LIN {X 0,Y 305.488,Z 300.056,A -85,B 0,C 180,E1 -15819.813,E2 -15819.813} C_VEL
LIN {X 0,Y 305.533,Z 300.043,A -85,B 0,C 180,E1 -15822.6,E2 -15822.6} C_VEL
LIN {X 0,Y 305.618,Z 300.037,A -85,B 0,C 180,E1 -15825.347,E2 -15825.347} C_VEL
LIN {X 0,Y 305.615,Z 300.039,A -85,B 0,C 180,E1 -15829.399,E2 -15829.399} C_VEL
LIN {X 0,Y 305.761,Z 300.017,A -85,B 0,C 180,E1 -15832.073,E2 -15832.073} C_VEL
LIN {X 0,Y 305.66,Z 300.028,A -85,B 0,C 180,E1 -15834.723,E2 -15834.723} C_VEL
LIN {X 0,Y 305.94,Z 299.998,A -85,B 0,C 180,E1 -15838.684,E2 -15838.684} C_VEL
LIN {X 0,Y 305.938,Z 299.999,A -85,B 0,C 180,E1 -15841.316,E2 -15841.316} C_VEL
LIN {X 0,Y 305.788,Z 300.021,A -85,B 0,C 180,E1 -15846.599,E2 -15846.599} C_VEL
LIN {X 0,Y 305.685,Z 300.023,A -85,B 0,C 180,E1 -15849.261,E2 -15849.261} C_VEL
LIN {X 0,Y 305.575,Z 300.037,A -85,B 0,C 180,E1 -15853.296,E2 -15853.296} C_VEL
LIN {X 0,Y 305.542,Z 300.054,A -85,B 0,C 180,E1 -15856.023,E2 -15856.023} C_VEL
LIN {X 0,Y 305.475,Z 300.064,A -85,B 0,C 180,E1 -15860.188,E2 -15860.188} C_VEL
LIN {X 0,Y 305.447,Z 300.063,A -85,B 0,C 180,E1 -15864.466,E2 -15864.466} C_VEL
LIN {X 0,Y 305.444,Z 300.063,A -85,B 0,C 180,E1 -15867.399,E2 -15867.399} C_VEL
LIN {X 0,Y 305.423,Z 300.065,A -85,B 0,C 180,E1 -15870.413,E2 -15870.413} C_VEL
LIN {X 0,Y 305.457,Z 300.057,A -85,B 0,C 180,E1 -15874.079,E2 -15874.079} C_VEL
LIN {X 0,Y 305.446,Z 300.057,A -85,B 0,C 180,E1 -15876.743,E2 -15876.743} C_VEL
LIN {X 0,Y 305.403,Z 300.042,A -85,B 0,C 180,E1 -15880.59,E2 -15880.59} C_VEL
LIN {X 0,Y 305.415,Z 300.065,A -85,B 0,C 180,E1 -15883.657,E2 -15883.657} C_VEL
LIN {X 0,Y 305.407,Z 300.074,A -85,B 0,C 180,E1 -15886.973,E2 -15886.973} C_VEL
LIN {X 0,Y 308.846,Z 311.457,A -85,B 0,C 180,E1 -15890.686,E2 -15890.686} C_VEL
LIN {X 0,Y 309.648,Z 314.272,A -85,B 0,C 180,E1 -15891.522,E2 -15891.522} C_VEL
LIN {X 0,Y 318.82,Z 331.707,A -85,B 0,C 180,E1 -15893.292,E2 -15893.292} C_VEL
LIN {X 0,Y 326.748,Z 348.767,A -85,B 0,C 180,E1 -15894.765,E2 -15894.765} C_VEL
LIN {X 0,Y 329.337,Z 355.038,A -85,B 0,C 180,E1 -15895.243,E2 -15895.243} C_VEL
LIN {X 0,Y 331.45,Z 367.704,A -85,B 0,C 180,E1 -15895.82,E2 -15895.82} C_VEL
LIN {X 0,Y 328.353,Z 458.786,A -85,B 0,C 180,E1 -15897.787,E2 -15897.787} C_VEL
LIN {X 0,Y 327.344,Z 483.079,A -85,B 0,C 180,E1 -15898.355,E2 -15898.355} C_VEL
LIN {X 0,Y 326.05,Z 498.482,A -85,B 0,C 180,E1 -15898.939,E2 -15898.939} C_VEL
LIN {X 0,Y 324.286,Z 513.373,A -85,B 0,C 180,E1 -15899.744,E2 -15899.744} C_VEL
LIN {X 0,Y 322.3,Z 527.368,A -85,B 0,C 180,E1 -15900.754,E2 -15900.754} C_VEL
LIN {X 0,Y 320.028,Z 540.986,A -85,B 0,C 180,E1 -15902.005,E2 -15902.005} C_VEL
LIN {X 0,Y 317.409,Z 554.417,A -85,B 0,C 180,E1 -15903.539,E2 -15903.539} C_VEL
LIN {X 0,Y 314.806,Z 566.654,A -85,B 0,C 180,E1 -15905.255,E2 -15905.255} C_VEL
LIN {X 0,Y 312.33,Z 578.002,A -85,B 0,C 180,E1 -15907.196,E2 -15907.196} C_VEL
LIN {X 0,Y 310.016,Z 588.691,A -85,B 0,C 180,E1 -15909.429,E2 -15909.429} C_VEL
LIN {X 0,Y 307.942,Z 597.734,A -85,B 0,C 180,E1 -15911.712,E2 -15911.712} C_VEL
LIN {X 0,Y 306.367,Z 605.243,A -85,B 0,C 180,E1 -15914.022,E2 -15914.022} C_VEL
LIN {X 0,Y 305.088,Z 612.254,A -85,B 0,C 180,E1 -15916.682,E2 -15916.682} C_VEL
LIN {X 0,Y 304.181,Z 617.769,A -85,B 0,C 180,E1 -15919.349,E2 -15919.349} C_VEL
LIN {X 0,Y 303.767,Z 621.945,A -85,B 0,C 180,E1 -15922.021,E2 -15922.021} C_VEL
LIN {X 0,Y 303.596,Z 624.875,A -85,B 0,C 180,E1 -15924.687,E2 -15924.687} C_VEL
LIN {X 0,Y 303.592,Z 626.624,A -85,B 0,C 180,E1 -15927.346,E2 -15927.346} C_VEL
LIN {X 0,Y 303.602,Z 627.222,A -85,B 0,C 180,E1 -15930,E2 -15930} C_VEL
LIN {X 0,Y 303.591,Z 626.615,A -85,B 0,C 180,E1 -15932.654,E2 -15932.654} C_VEL
LIN {X 0,Y 303.624,Z 624.655,A -85,B 0,C 180,E1 -15935.544,E2 -15935.544} C_VEL
LIN {X 0,Y 303.765,Z 621.916,A -85,B 0,C 180,E1 -15937.979,E2 -15937.979} C_VEL
LIN {X 0,Y 304.18,Z 617.735,A -85,B 0,C 180,E1 -15940.651,E2 -15940.651} C_VEL
LIN {X 0,Y 305.08,Z 612.205,A -85,B 0,C 180,E1 -15943.318,E2 -15943.318} C_VEL
LIN {X 0,Y 306.362,Z 605.173,A -85,B 0,C 180,E1 -15945.978,E2 -15945.978} C_VEL
LIN {X 0,Y 308.205,Z 596.433,A -85,B 0,C 180,E1 -15948.617,E2 -15948.617} C_VEL
LIN {X 0,Y 310.357,Z 587.156,A -85,B 0,C 180,E1 -15950.894,E2 -15950.894} C_VEL
LIN {X 0,Y 312.379,Z 577.896,A -85,B 0,C 180,E1 -15952.8,E2 -15952.8} C_VEL
LIN {X 0,Y 314.82,Z 566.53,A -85,B 0,C 180,E1 -15954.744,E2 -15954.744} C_VEL
LIN {X 0,Y 317.413,Z 554.269,A -85,B 0,C 180,E1 -15956.461,E2 -15956.461} C_VEL
LIN {X 0,Y 320.015,Z 540.79,A -85,B 0,C 180,E1 -15957.996,E2 -15957.996} C_VEL
LIN {X 0,Y 322.452,Z 526.115,A -85,B 0,C 180,E1 -15959.33,E2 -15959.33} C_VEL
LIN {X 0,Y 324.573,Z 510.682,A -85,B 0,C 180,E1 -15960.406,E2 -15960.406} C_VEL
LIN {X 0,Y 326.261,Z 495.632,A -85,B 0,C 180,E1 -15961.174,E2 -15961.174} C_VEL
LIN {X 0,Y 327.451,Z 479.865,A -85,B 0,C 180,E1 -15961.724,E2 -15961.724} C_VEL
LIN {X 0,Y 330.751,Z 387.93,A -85,B 0,C 180,E1 -15963.718,E2 -15963.718} C_VEL
LIN {X 0,Y 331.325,Z 367.172,A -85,B 0,C 180,E1 -15964.182,E2 -15964.182} C_VEL
LIN {X 0,Y 328.976,Z 353.98,A -85,B 0,C 180,E1 -15964.8,E2 -15964.8} C_VEL
LIN {X 0,Y 320.543,Z 335.198,A -85,B 0,C 180,E1 -15966.354,E2 -15966.354} C_VEL
LIN {X 0,Y 311.857,Z 318.359,A -85,B 0,C 180,E1 -15968.007,E2 -15968.007} C_VEL
LIN {X 0,Y 309.559,Z 314.082,A -85,B 0,C 180,E1 -15968.469,E2 -15968.469} C_VEL
LIN {X 0,Y 306.242,Z 302.692,A -85,B 0,C 180,E1 -15972.101,E2 -15972.101} C_VEL
LIN {X 0,Y 305.408,Z 300.068,A -85,B 0,C 180,E1 -15973.027,E2 -15973.027} C_VEL
LIN {X 0,Y 305.429,Z 300.063,A -85,B 0,C 180,E1 -15977.418,E2 -15977.418} C_VEL
LIN {X 0,Y 305.439,Z 300.06,A -85,B 0,C 180,E1 -15981.592,E2 -15981.592} C_VEL
LIN {X 0,Y 305.453,Z 300.057,A -85,B 0,C 180,E1 -15984.886,E2 -15984.886} C_VEL
LIN {X 0,Y 305.434,Z 300.063,A -85,B 0,C 180,E1 -15988.358,E2 -15988.358} C_VEL
LIN {X 0,Y 305.467,Z 300.058,A -85,B 0,C 180,E1 -15991.108,E2 -15991.108} C_VEL
LIN {X 0,Y 305.472,Z 300.06,A -85,B 0,C 180,E1 -15994.079,E2 -15994.079} C_VEL
LIN {X 0,Y 305.455,Z 300.059,A -85,B 0,C 180,E1 -15998.4,E2 -15998.4} C_VEL
LIN {X 0,Y 305.529,Z 300.035,A -85,B 0,C 180,E1 -16002.6,E2 -16002.6} C_VEL
LIN {X 0,Y 305.618,Z 300.04,A -85,B 0,C 180,E1 -16005.348,E2 -16005.348} C_VEL
LIN {X 0,Y 305.612,Z 300.009,A -85,B 0,C 180,E1 -16009.399,E2 -16009.399} C_VEL
LIN {X 0,Y 305.732,Z 300.027,A -85,B 0,C 180,E1 -16012.072,E2 -16012.072} C_VEL
LIN {X 0,Y 305.651,Z 300.027,A -85,B 0,C 180,E1 -16014.723,E2 -16014.723} C_VEL
LIN {X 0,Y 305.938,Z 299.991,A -85,B 0,C 180,E1 -16018.684,E2 -16018.684} C_VEL
LIN {X 0,Y 305.926,Z 300.001,A -85,B 0,C 180,E1 -16021.317,E2 -16021.317} C_VEL
LIN {X 0,Y 305.658,Z 300.036,A -85,B 0,C 180,E1 -16025.277,E2 -16025.277} C_VEL
LIN {X 0,Y 305.753,Z 300.023,A -85,B 0,C 180,E1 -16027.927,E2 -16027.927} C_VEL
LIN {X 0,Y 305.588,Z 300.043,A -85,B 0,C 180,E1 -16031.946,E2 -16031.946} C_VEL
LIN {X 0,Y 305.6,Z 300.036,A -85,B 0,C 180,E1 -16035.014,E2 -16035.014} C_VEL
LIN {X 0,Y 305.509,Z 300.039,A -85,B 0,C 180,E1 -16038.788,E2 -16038.788} C_VEL
LIN {X 0,Y 305.479,Z 300.052,A -85,B 0,C 180,E1 -16043.04,E2 -16043.04} C_VEL
LIN {X 0,Y 305.497,Z 300.038,A -85,B 0,C 180,E1 -16046.211,E2 -16046.211} C_VEL
LIN {X 0,Y 305.478,Z 300.046,A -85,B 0,C 180,E1 -16049.047,E2 -16049.047} C_VEL
LIN {X 0,Y 305.436,Z 300.057,A -85,B 0,C 180,E1 -16051.953,E2 -16051.953} C_VEL
LIN {X 0,Y 305.455,Z 300.057,A -85,B 0,C 180,E1 -16055.114,E2 -16055.114} C_VEL
LIN {X 0,Y 305.434,Z 300.061,A -85,B 0,C 180,E1 -16058.527,E2 -16058.527} C_VEL
LIN {X 0,Y 305.45,Z 300.058,A -85,B 0,C 180,E1 -16062.587,E2 -16062.587} C_VEL
LIN {X 0,Y 305.421,Z 300.065,A -85,B 0,C 180,E1 -16066.346,E2 -16066.346} C_VEL
LIN {X 0,Y 305.455,Z 300.061,A -85,B 0,C 180,E1 -16069.893,E2 -16069.893} C_VEL
LIN {X 0,Y 305.446,Z 300.076,A -85,B 0,C 180,E1 -16070.761,E2 -16070.761} C_VEL
LIN {X 0,Y 305.611,Z 300.81,A -85,B 0,C 180,E1 -16071.007,E2 -16071.007} C_VEL
LIN {X 0,Y 306.858,Z 303.478,A -85,B 0,C 180,E1 -16071.275,E2 -16071.275} C_VEL
LIN {X 0,Y 308.864,Z 306.49,A -85,B 0,C 180,E1 -16071.663,E2 -16071.663} C_VEL
LIN {X 0,Y 314.538,Z 316.113,A -85,B 0,C 180,E1 -16072.754,E2 -16072.754} C_VEL
LIN {X 0,Y 323.344,Z 332.892,A -85,B 0,C 180,E1 -16074.393,E2 -16074.393} C_VEL
LIN {X 0,Y 331.832,Z 351.222,A -85,B 0,C 180,E1 -16075.916,E2 -16075.916} C_VEL
LIN {X 0,Y 329.184,Z 429.846,A -85,B 0,C 180,E1 -16077.619,E2 -16077.619} C_VEL
LIN {X 0,Y 327.853,Z 465.342,A -85,B 0,C 180,E1 -16078.41,E2 -16078.41} C_VEL
LIN {X 0,Y 326.688,Z 481.055,A -85,B 0,C 180,E1 -16078.99,E2 -16078.99} C_VEL
LIN {X 0,Y 325.166,Z 496.001,A -85,B 0,C 180,E1 -16079.798,E2 -16079.798} C_VEL
LIN {X 0,Y 323.552,Z 509.183,A -85,B 0,C 180,E1 -16080.75,E2 -16080.75} C_VEL
LIN {X 0,Y 321.363,Z 522.677,A -85,B 0,C 180,E1 -16081.954,E2 -16081.954} C_VEL
LIN {X 0,Y 319.149,Z 535.149,A -85,B 0,C 180,E1 -16083.342,E2 -16083.342} C_VEL
LIN {X 0,Y 316.521,Z 547.786,A -85,B 0,C 180,E1 -16085.048,E2 -16085.048} C_VEL
LIN {X 0,Y 314.516,Z 557.561,A -85,B 0,C 180,E1 -16086.652,E2 -16086.652} C_VEL
LIN {X 0,Y 312.254,Z 567.396,A -85,B 0,C 180,E1 -16088.547,E2 -16088.547} C_VEL
LIN {X 0,Y 310.023,Z 577.09,A -85,B 0,C 180,E1 -16090.81,E2 -16090.81} C_VEL
LIN {X 0,Y 308.026,Z 585.389,A -85,B 0,C 180,E1 -16093.163,E2 -16093.163} C_VEL
LIN {X 0,Y 306.706,Z 591.827,A -85,B 0,C 180,E1 -16095.401,E2 -16095.401} C_VEL
LIN {X 0,Y 305.372,Z 597.993,A -85,B 0,C 180,E1 -16098.046,E2 -16098.046} C_VEL
LIN {X 0,Y 304.57,Z 602.747,A -85,B 0,C 180,E1 -16100.705,E2 -16100.705} C_VEL
LIN {X 0,Y 304.046,Z 606.228,A -85,B 0,C 180,E1 -16103.363,E2 -16103.363} C_VEL
LIN {X 0,Y 303.789,Z 608.528,A -85,B 0,C 180,E1 -16106.02,E2 -16106.02} C_VEL
LIN {X 0,Y 303.608,Z 609.703,A -85,B 0,C 180,E1 -16108.674,E2 -16108.674} C_VEL
LIN {X 0,Y 303.608,Z 609.717,A -85,B 0,C 180,E1 -16111.326,E2 -16111.326} C_VEL
LIN {X 0,Y 303.781,Z 608.598,A -85,B 0,C 180,E1 -16113.98,E2 -16113.98} C_VEL
LIN {X 0,Y 304.041,Z 606.352,A -85,B 0,C 180,E1 -16116.637,E2 -16116.637} C_VEL
LIN {X 0,Y 304.55,Z 602.921,A -85,B 0,C 180,E1 -16119.296,E2 -16119.296} C_VEL
LIN {X 0,Y 305.337,Z 598.223,A -85,B 0,C 180,E1 -16121.955,E2 -16121.955} C_VEL
LIN {X 0,Y 306.679,Z 592.126,A -85,B 0,C 180,E1 -16124.6,E2 -16124.6} C_VEL
LIN {X 0,Y 308.302,Z 584.452,A -85,B 0,C 180,E1 -16127.238,E2 -16127.238} C_VEL
LIN {X 0,Y 310.219,Z 576.262,A -85,B 0,C 180,E1 -16129.521,E2 -16129.521} C_VEL
LIN {X 0,Y 312.519,Z 566.392,A -85,B 0,C 180,E1 -16131.78,E2 -16131.78} C_VEL
LIN {X 0,Y 314.726,Z 556.192,A -85,B 0,C 180,E1 -16133.715,E2 -16133.715} C_VEL
LIN {X 0,Y 317.365,Z 544.212,A -85,B 0,C 180,E1 -16135.583,E2 -16135.583} C_VEL
LIN {X 0,Y 319.716,Z 532.118,A -85,B 0,C 180,E1 -16137.137,E2 -16137.137} C_VEL
LIN {X 0,Y 322.078,Z 518.969,A -85,B 0,C 180,E1 -16138.51,E2 -16138.51} C_VEL
LIN {X 0,Y 324.033,Z 505.698,A -85,B 0,C 180,E1 -16139.632,E2 -16139.632} C_VEL
LIN {X 0,Y 325.667,Z 491.769,A -85,B 0,C 180,E1 -16140.561,E2 -16140.561} C_VEL
LIN {X 0,Y 327.101,Z 476.492,A -85,B 0,C 180,E1 -16141.31,E2 -16141.31} C_VEL
LIN {X 0,Y 328.115,Z 461.755,A -85,B 0,C 180,E1 -16141.787,E2 -16141.787} C_VEL
LIN {X 0,Y 331.406,Z 368.205,A -85,B 0,C 180,E1 -16143.815,E2 -16143.815} C_VEL
LIN {X 0,Y 331.011,Z 364.38,A -85,B 0,C 180,E1 -16143.96,E2 -16143.96} C_VEL
LIN {X 0,Y 329.874,Z 360.802,A -85,B 0,C 180,E1 -16144.186,E2 -16144.186} C_VEL
LIN {X 0,Y 324.321,Z 349.64,A -85,B 0,C 180,E1 -16145.156,E2 -16145.156} C_VEL
LIN {X 0,Y 316.974,Z 334.175,A -85,B 0,C 180,E1 -16146.53,E2 -16146.53} C_VEL
LIN {X 0,Y 309.997,Z 320.812,A -85,B 0,C 180,E1 -16147.881,E2 -16147.881} C_VEL
LIN {X 0,Y 303.322,Z 309.395,A -85,B 0,C 180,E1 -16149.217,E2 -16149.217} C_VEL
LIN {X 0,Y 301.13,Z 305.909,A -85,B 0,C 180,E1 -16149.667,E2 -16149.667} C_VEL
LIN {X 0,Y 298.982,Z 302.953,A -85,B 0,C 180,E1 -16150.102,E2 -16150.102} C_VEL
LIN {X 0,Y 298.409,Z 300.93,A -85,B 0,C 180,E1 -16150.301,E2 -16150.301} C_VEL
LIN {X 0,Y 298.396,Z 300.94,A -85,B 0,C 180,E1 -16153.102,E2 -16153.102} C_VEL
LIN {X 0,Y 298.399,Z 300.931,A -85,B 0,C 180,E1 -16156.92,E2 -16156.92} C_VEL
LIN {X 0,Y 298.393,Z 300.941,A -85,B 0,C 180,E1 -16161.007,E2 -16161.007} C_VEL
LIN {X 0,Y 298.399,Z 300.919,A -85,B 0,C 180,E1 -16163.927,E2 -16163.927} C_VEL
LIN {X 0,Y 298.387,Z 300.935,A -85,B 0,C 180,E1 -16167.199,E2 -16167.199} C_VEL
LIN {X 0,Y 298.408,Z 300.919,A -85,B 0,C 180,E1 -16170.62,E2 -16170.62} C_VEL
LIN {X 0,Y 298.438,Z 300.932,A -85,B 0,C 180,E1 -16173.489,E2 -16173.489} C_VEL
LIN {X 0,Y 298.422,Z 300.939,A -85,B 0,C 180,E1 -16176.7,E2 -16176.7} C_VEL
LIN {X 0,Y 298.496,Z 300.929,A -85,B 0,C 180,E1 -16180.754,E2 -16180.754} C_VEL
LIN {X 0,Y 298.579,Z 300.917,A -85,B 0,C 180,E1 -16184.994,E2 -16184.994} C_VEL
LIN {X 0,Y 298.574,Z 300.918,A -85,B 0,C 180,E1 -16189.146,E2 -16189.146} C_VEL
LIN {X 0,Y 298.708,Z 300.896,A -85,B 0,C 180,E1 -16191.884,E2 -16191.884} C_VEL
LIN {X 0,Y 298.63,Z 300.905,A -85,B 0,C 180,E1 -16194.598,E2 -16194.598} C_VEL
LIN {X 0,Y 298.907,Z 300.874,A -85,B 0,C 180,E1 -16198.653,E2 -16198.653} C_VEL
LIN {X 0,Y 298.905,Z 300.875,A -85,B 0,C 180,E1 -16201.347,E2 -16201.347} C_VEL
LIN {X 0,Y 298.737,Z 300.901,A -85,B 0,C 180,E1 -16206.755,E2 -16206.755} C_VEL
LIN {X 0,Y 298.616,Z 300.904,A -85,B 0,C 180,E1 -16209.482,E2 -16209.482} C_VEL
LIN {X 0,Y 298.534,Z 300.914,A -85,B 0,C 180,E1 -16213.616,E2 -16213.616} C_VEL
LIN {X 0,Y 298.475,Z 300.931,A -85,B 0,C 180,E1 -16216.413,E2 -16216.413} C_VEL
LIN {X 0,Y 298.433,Z 300.938,A -85,B 0,C 180,E1 -16219.617,E2 -16219.617} C_VEL
LIN {X 0,Y 298.38,Z 300.944,A -85,B 0,C 180,E1 -16223.604,E2 -16223.604} C_VEL
LIN {X 0,Y 298.395,Z 300.936,A -85,B 0,C 180,E1 -16226.583,E2 -16226.583} C_VEL
LIN {X 0,Y 298.386,Z 300.943,A -85,B 0,C 180,E1 -16229.645,E2 -16229.645} C_VEL
LIN {X 0,Y 298.385,Z 300.933,A -85,B 0,C 180,E1 -16232.801,E2 -16232.801} C_VEL
LIN {X 0,Y 298.42,Z 300.932,A -85,B 0,C 180,E1 -16236.803,E2 -16236.803} C_VEL
LIN {X 0,Y 298.341,Z 300.923,A -85,B 0,C 180,E1 -16241.269,E2 -16241.269} C_VEL
LIN {X 0,Y 298.35,Z 300.947,A -85,B 0,C 180,E1 -16245.036,E2 -16245.036} C_VEL
LIN {X 0,Y 298.373,Z 300.96,A -85,B 0,C 180,E1 -16246.044,E2 -16246.044} C_VEL
LIN {X 0,Y 301.739,Z 312.035,A -85,B 0,C 180,E1 -16249.807,E2 -16249.807} C_VEL
LIN {X 0,Y 302.287,Z 313.971,A -85,B 0,C 180,E1 -16250.402,E2 -16250.402} C_VEL
LIN {X 0,Y 310.364,Z 328.922,A -85,B 0,C 180,E1 -16252.047,E2 -16252.047} C_VEL
LIN {X 0,Y 318.508,Z 345.475,A -85,B 0,C 180,E1 -16253.628,E2 -16253.628} C_VEL
LIN {X 0,Y 323.829,Z 358.27,A -85,B 0,C 180,E1 -16254.655,E2 -16254.655} C_VEL
LIN {X 0,Y 325.57,Z 369.904,A -85,B 0,C 180,E1 -16255.177,E2 -16255.177} C_VEL
LIN {X 0,Y 321.691,Z 476.003,A -85,B 0,C 180,E1 -16257.501,E2 -16257.501} C_VEL
LIN {X 0,Y 320.646,Z 491.352,A -85,B 0,C 180,E1 -16257.986,E2 -16257.986} C_VEL
LIN {X 0,Y 319.142,Z 505.626,A -85,B 0,C 180,E1 -16258.651,E2 -16258.651} C_VEL
LIN {X 0,Y 317.264,Z 519.739,A -85,B 0,C 180,E1 -16259.547,E2 -16259.547} C_VEL
LIN {X 0,Y 315.181,Z 532.909,A -85,B 0,C 180,E1 -16260.623,E2 -16260.623} C_VEL
LIN {X 0,Y 312.612,Z 546.5,A -85,B 0,C 180,E1 -16262.012,E2 -16262.012} C_VEL
LIN {X 0,Y 310.005,Z 558.926,A -85,B 0,C 180,E1 -16263.583,E2 -16263.583} C_VEL
LIN {X 0,Y 307.417,Z 570.373,A -85,B 0,C 180,E1 -16265.341,E2 -16265.341} C_VEL
LIN {X 0,Y 304.917,Z 581.187,A -85,B 0,C 180,E1 -16267.352,E2 -16267.352} C_VEL
LIN {X 0,Y 302.975,Z 589.85,A -85,B 0,C 180,E1 -16269.284,E2 -16269.284} C_VEL
LIN {X 0,Y 300.864,Z 598.656,A -85,B 0,C 180,E1 -16271.619,E2 -16271.619} C_VEL
LIN {X 0,Y 299.142,Z 606.68,A -85,B 0,C 180,E1 -16274.234,E2 -16274.234} C_VEL
LIN {X 0,Y 297.858,Z 613.546,A -85,B 0,C 180,E1 -16277.047,E2 -16277.047} C_VEL
LIN {X 0,Y 297.019,Z 618.735,A -85,B 0,C 180,E1 -16279.778,E2 -16279.778} C_VEL
LIN {X 0,Y 296.694,Z 621.742,A -85,B 0,C 180,E1 -16281.829,E2 -16281.829} C_VEL
LIN {X 0,Y 296.511,Z 624.672,A -85,B 0,C 180,E1 -16284.56,E2 -16284.56} C_VEL
LIN {X 0,Y 296.516,Z 626.422,A -85,B 0,C 180,E1 -16287.283,E2 -16287.283} C_VEL
LIN {X 0,Y 296.517,Z 627.019,A -85,B 0,C 180,E1 -16290,E2 -16290} C_VEL
LIN {X 0,Y 296.515,Z 626.412,A -85,B 0,C 180,E1 -16292.717,E2 -16292.717} C_VEL
LIN {X 0,Y 296.511,Z 624.65,A -85,B 0,C 180,E1 -16295.44,E2 -16295.44} C_VEL
LIN {X 0,Y 296.691,Z 621.711,A -85,B 0,C 180,E1 -16298.171,E2 -16298.171} C_VEL
LIN {X 0,Y 297.142,Z 617.529,A -85,B 0,C 180,E1 -16300.907,E2 -16300.907} C_VEL
LIN {X 0,Y 298.089,Z 611.998,A -85,B 0,C 180,E1 -16303.637,E2 -16303.637} C_VEL
LIN {X 0,Y 299.481,Z 604.967,A -85,B 0,C 180,E1 -16306.356,E2 -16306.356} C_VEL
LIN {X 0,Y 301.407,Z 596.226,A -85,B 0,C 180,E1 -16309.052,E2 -16309.052} C_VEL
LIN {X 0,Y 303.674,Z 586.949,A -85,B 0,C 180,E1 -16311.377,E2 -16311.377} C_VEL
LIN {X 0,Y 305.806,Z 577.519,A -85,B 0,C 180,E1 -16313.355,E2 -16313.355} C_VEL
LIN {X 0,Y 308.362,Z 566.323,A -85,B 0,C 180,E1 -16315.298,E2 -16315.298} C_VEL
LIN {X 0,Y 311.011,Z 554.061,A -85,B 0,C 180,E1 -16317.049,E2 -16317.049} C_VEL
LIN {X 0,Y 313.737,Z 540.582,A -85,B 0,C 180,E1 -16318.607,E2 -16318.607} C_VEL
LIN {X 0,Y 316.072,Z 527.027,A -85,B 0,C 180,E1 -16319.868,E2 -16319.868} C_VEL
LIN {X 0,Y 318.296,Z 511.725,A -85,B 0,C 180,E1 -16320.979,E2 -16320.979} C_VEL
LIN {X 0,Y 320.122,Z 496.31,A -85,B 0,C 180,E1 -16321.795,E2 -16321.795} C_VEL
LIN {X 0,Y 321.388,Z 481.073,A -85,B 0,C 180,E1 -16322.348,E2 -16322.348} C_VEL
LIN {X 0,Y 324.853,Z 387.706,A -85,B 0,C 180,E1 -16324.415,E2 -16324.415} C_VEL
LIN {X 0,Y 325.441,Z 368.299,A -85,B 0,C 180,E1 -16324.853,E2 -16324.853} C_VEL
LIN {X 0,Y 323.377,Z 356.804,A -85,B 0,C 180,E1 -16325.411,E2 -16325.411} C_VEL
LIN {X 0,Y 315.248,Z 338.65,A -85,B 0,C 180,E1 -16326.964,E2 -16326.964} C_VEL
LIN {X 0,Y 307.169,Z 322.776,A -85,B 0,C 180,E1 -16328.559,E2 -16328.559} C_VEL
LIN {X 0,Y 302.237,Z 313.763,A -85,B 0,C 180,E1 -16329.595,E2 -16329.595} C_VEL
LIN {X 0,Y 298.929,Z 302.989,A -85,B 0,C 180,E1 -16333.212,E2 -16333.212} C_VEL
LIN {X 0,Y 298.356,Z 300.949,A -85,B 0,C 180,E1 -16333.953,E2 -16333.953} C_VEL
LIN {X 0,Y 298.365,Z 300.944,A -85,B 0,C 180,E1 -16336.914,E2 -16336.914} C_VEL
LIN {X 0,Y 298.347,Z 300.947,A -85,B 0,C 180,E1 -16341.018,E2 -16341.018} C_VEL
LIN {X 0,Y 298.397,Z 300.936,A -85,B 0,C 180,E1 -16343.927,E2 -16343.927} C_VEL
LIN {X 0,Y 298.385,Z 300.935,A -85,B 0,C 180,E1 -16347.199,E2 -16347.199} C_VEL
LIN {X 0,Y 298.394,Z 300.938,A -85,B 0,C 180,E1 -16350.625,E2 -16350.625} C_VEL
LIN {X 0,Y 298.406,Z 300.939,A -85,B 0,C 180,E1 -16354.917,E2 -16354.917} C_VEL
LIN {X 0,Y 298.386,Z 300.942,A -85,B 0,C 180,E1 -16357.861,E2 -16357.861} C_VEL
LIN {X 0,Y 298.455,Z 300.903,A -85,B 0,C 180,E1 -16360.751,E2 -16360.751} C_VEL
LIN {X 0,Y 298.578,Z 300.918,A -85,B 0,C 180,E1 -16364.994,E2 -16364.994} C_VEL
LIN {X 0,Y 298.571,Z 300.883,A -85,B 0,C 180,E1 -16369.146,E2 -16369.146} C_VEL
LIN {X 0,Y 298.678,Z 300.907,A -85,B 0,C 180,E1 -16371.884,E2 -16371.884} C_VEL
LIN {X 0,Y 298.621,Z 300.902,A -85,B 0,C 180,E1 -16374.598,E2 -16374.598} C_VEL
LIN {X 0,Y 298.904,Z 300.867,A -85,B 0,C 180,E1 -16378.653,E2 -16378.653} C_VEL
LIN {X 0,Y 298.894,Z 300.877,A -85,B 0,C 180,E1 -16381.347,E2 -16381.347} C_VEL
LIN {X 0,Y 298.738,Z 300.89,A -85,B 0,C 180,E1 -16386.755,E2 -16386.755} C_VEL
LIN {X 0,Y 298.617,Z 300.912,A -85,B 0,C 180,E1 -16389.483,E2 -16389.483} C_VEL
LIN {X 0,Y 298.535,Z 300.921,A -85,B 0,C 180,E1 -16393.616,E2 -16393.616} C_VEL
LIN {X 0,Y 298.476,Z 300.929,A -85,B 0,C 180,E1 -16396.413,E2 -16396.413} C_VEL
LIN {X 0,Y 298.438,Z 300.908,A -85,B 0,C 180,E1 -16399.619,E2 -16399.619} C_VEL
LIN {X 0,Y 298.418,Z 300.939,A -85,B 0,C 180,E1 -16403.601,E2 -16403.601} C_VEL
LIN {X 0,Y 298.449,Z 300.911,A -85,B 0,C 180,E1 -16406.578,E2 -16406.578} C_VEL
LIN {X 0,Y 298.409,Z 300.935,A -85,B 0,C 180,E1 -16409.642,E2 -16409.642} C_VEL
LIN {X 0,Y 298.389,Z 300.938,A -85,B 0,C 180,E1 -16412.801,E2 -16412.801} C_VEL
LIN {X 0,Y 298.438,Z 300.933,A -85,B 0,C 180,E1 -16416.808,E2 -16416.808} C_VEL
LIN {X 0,Y 298.383,Z 300.942,A -85,B 0,C 180,E1 -16421.089,E2 -16421.089} C_VEL
LIN {X 0,Y 298.395,Z 300.939,A -85,B 0,C 180,E1 -16423.104,E2 -16423.104} C_VEL
LIN {X 0,Y 298.4,Z 300.939,A -85,B 0,C 180,E1 -16426.922,E2 -16426.922} C_VEL
LIN {X 0,Y 298.433,Z 301.075,A -85,B 0,C 180,E1 -16429.881,E2 -16429.881} C_VEL
LIN {X 0,Y 299.531,Z 303.971,A -85,B 0,C 180,E1 -16430.148,E2 -16430.148} C_VEL
LIN {X 0,Y 301.217,Z 306.064,A -85,B 0,C 180,E1 -16430.481,E2 -16430.481} C_VEL
LIN {X 0,Y 303.329,Z 309.406,A -85,B 0,C 180,E1 -16430.912,E2 -16430.912} C_VEL
LIN {X 0,Y 310.704,Z 322.089,A -85,B 0,C 180,E1 -16432.382,E2 -16432.382} C_VEL
LIN {X 0,Y 319.358,Z 338.976,A -85,B 0,C 180,E1 -16434.041,E2 -16434.041} C_VEL
LIN {X 0,Y 325.934,Z 353.415,A -85,B 0,C 180,E1 -16435.263,E2 -16435.263} C_VEL
LIN {X 0,Y 322.747,Z 443.895,A -85,B 0,C 180,E1 -16437.25,E2 -16437.25} C_VEL
LIN {X 0,Y 321.667,Z 467.854,A -85,B 0,C 180,E1 -16437.822,E2 -16437.822} C_VEL
LIN {X 0,Y 320.514,Z 482.523,A -85,B 0,C 180,E1 -16438.401,E2 -16438.401} C_VEL
LIN {X 0,Y 318.933,Z 497.124,A -85,B 0,C 180,E1 -16439.219,E2 -16439.219} C_VEL
LIN {X 0,Y 317.067,Z 511.471,A -85,B 0,C 180,E1 -16440.296,E2 -16440.296} C_VEL
LIN {X 0,Y 314.826,Z 524.44,A -85,B 0,C 180,E1 -16441.501,E2 -16441.501} C_VEL
LIN {X 0,Y 312.31,Z 537.89,A -85,B 0,C 180,E1 -16443.072,E2 -16443.072} C_VEL
LIN {X 0,Y 309.608,Z 550.292,A -85,B 0,C 180,E1 -16444.847,E2 -16444.847} C_VEL
LIN {X 0,Y 307.805,Z 558.585,A -85,B 0,C 180,E1 -16446.277,E2 -16446.277} C_VEL
LIN {X 0,Y 305.249,Z 569.078,A -85,B 0,C 180,E1 -16448.385,E2 -16448.385} C_VEL
LIN {X 0,Y 303.004,Z 578.517,A -85,B 0,C 180,E1 -16450.7,E2 -16450.7} C_VEL
LIN {X 0,Y 300.841,Z 587.164,A -85,B 0,C 180,E1 -16453.298,E2 -16453.298} C_VEL
LIN {X 0,Y 299.45,Z 593.701,A -85,B 0,C 180,E1 -16455.734,E2 -16455.734} C_VEL
LIN {X 0,Y 298.152,Z 599.514,A -85,B 0,C 180,E1 -16458.442,E2 -16458.442} C_VEL
LIN {X 0,Y 297.534,Z 602.952,A -85,B 0,C 180,E1 -16460.483,E2 -16460.483} C_VEL
LIN {X 0,Y 296.999,Z 606.432,A -85,B 0,C 180,E1 -16463.205,E2 -16463.205} C_VEL
LIN {X 0,Y 296.705,Z 608.732,A -85,B 0,C 180,E1 -16465.925,E2 -16465.925} C_VEL
LIN {X 0,Y 296.527,Z 609.906,A -85,B 0,C 180,E1 -16468.642,E2 -16468.642} C_VEL
LIN {X 0,Y 296.527,Z 609.919,A -85,B 0,C 180,E1 -16471.358,E2 -16471.358} C_VEL
LIN {X 0,Y 296.697,Z 608.801,A -85,B 0,C 180,E1 -16474.075,E2 -16474.075} C_VEL
LIN {X 0,Y 296.963,Z 606.556,A -85,B 0,C 180,E1 -16476.796,E2 -16476.796} C_VEL
LIN {X 0,Y 297.516,Z 603.124,A -85,B 0,C 180,E1 -16479.518,E2 -16479.518} C_VEL
LIN {X 0,Y 298.349,Z 598.426,A -85,B 0,C 180,E1 -16482.24,E2 -16482.24} C_VEL
LIN {X 0,Y 299.779,Z 592.329,A -85,B 0,C 180,E1 -16484.944,E2 -16484.944} C_VEL
LIN {X 0,Y 301.478,Z 584.654,A -85,B 0,C 180,E1 -16487.641,E2 -16487.641} C_VEL
LIN {X 0,Y 303.495,Z 576.464,A -85,B 0,C 180,E1 -16489.972,E2 -16489.972} C_VEL
LIN {X 0,Y 305.908,Z 566.593,A -85,B 0,C 180,E1 -16492.276,E2 -16492.276} C_VEL
LIN {X 0,Y 308.204,Z 556.473,A -85,B 0,C 180,E1 -16494.233,E2 -16494.233} C_VEL
LIN {X 0,Y 310.957,Z 544.412,A -85,B 0,C 180,E1 -16496.149,E2 -16496.149} C_VEL
LIN {X 0,Y 313.412,Z 532.317,A -85,B 0,C 180,E1 -16497.729,E2 -16497.729} C_VEL
LIN {X 0,Y 315.846,Z 519.167,A -85,B 0,C 180,E1 -16499.126,E2 -16499.126} C_VEL
LIN {X 0,Y 318.009,Z 504.924,A -85,B 0,C 180,E1 -16500.341,E2 -16500.341} C_VEL
LIN {X 0,Y 319.807,Z 490.007,A -85,B 0,C 180,E1 -16501.322,E2 -16501.322} C_VEL
LIN {X 0,Y 321.231,Z 474.854,A -85,B 0,C 180,E1 -16502.042,E2 -16502.042} C_VEL
LIN {X 0,Y 322.264,Z 458.931,A -85,B 0,C 180,E1 -16502.527,E2 -16502.527} C_VEL
LIN {X 0,Y 326.002,Z 353.448,A -85,B 0,C 180,E1 -16504.846,E2 -16504.846} C_VEL
LIN {X 0,Y 324.321,Z 349.64,A -85,B 0,C 180,E1 -16505.156,E2 -16505.156} C_VEL
LIN {X 0,Y 322.681,Z 346.474,A -85,B 0,C 180,E1 -16505.447,E2 -16505.447} C_VEL
LIN {X 0,Y 319.53,Z 342.389,A -85,B 0,C 180,E1 -16505.965,E2 -16505.965} C_VEL
LIN {X 0,Y 311.161,Z 334.1,A -85,B 0,C 180,E1 -16507.334,E2 -16507.334} C_VEL
LIN {X 0,Y 308.006,Z 330.062,A -85,B 0,C 180,E1 -16507.903,E2 -16507.903} C_VEL
LIN {X 0,Y 307.119,Z 328.545,A -85,B 0,C 180,E1 -16508.077,E2 -16508.077} C_VEL
LIN {X 0,Y 300.052,Z 316.063,A -85,B 0,C 180,E1 -16509.529,E2 -16509.529} C_VEL
LIN {X 0,Y 295.697,Z 309.483,A -85,B 0,C 180,E1 -16510.439,E2 -16510.439} C_VEL
LIN {X 0,Y 293.663,Z 306.233,A -85,B 0,C 180,E1 -16510.883,E2 -16510.883} C_VEL
LIN {X 0,Y 291.935,Z 303.863,A -85,B 0,C 180,E1 -16511.255,E2 -16511.255} C_VEL
LIN {X 0,Y 291.329,Z 301.817,A -85,B 0,C 180,E1 -16511.438,E2 -16511.438} C_VEL
LIN {X 0,Y 291.287,Z 301.826,A -85,B 0,C 180,E1 -16515.597,E2 -16515.597} C_VEL
LIN {X 0,Y 291.327,Z 301.808,A -85,B 0,C 180,E1 -16519.356,E2 -16519.356} C_VEL
LIN {X 0,Y 291.388,Z 301.791,A -85,B 0,C 180,E1 -16522.916,E2 -16522.916} C_VEL
LIN {X 0,Y 291.338,Z 301.82,A -85,B 0,C 180,E1 -16526.301,E2 -16526.301} C_VEL
LIN {X 0,Y 291.366,Z 301.791,A -85,B 0,C 180,E1 -16530.265,E2 -16530.265} C_VEL
LIN {X 0,Y 291.38,Z 301.807,A -85,B 0,C 180,E1 -16534.268,E2 -16534.268} C_VEL
LIN {X 0,Y 291.362,Z 301.812,A -85,B 0,C 180,E1 -16537.298,E2 -16537.298} C_VEL
LIN {X 0,Y 291.433,Z 301.808,A -85,B 0,C 180,E1 -16540.268,E2 -16540.268} C_VEL
LIN {X 0,Y 291.49,Z 301.803,A -85,B 0,C 180,E1 -16544.665,E2 -16544.665} C_VEL
LIN {X 0,Y 291.52,Z 301.799,A -85,B 0,C 180,E1 -16548.88,E2 -16548.88} C_VEL
LIN {X 0,Y 291.658,Z 301.772,A -85,B 0,C 180,E1 -16551.687,E2 -16551.687} C_VEL
LIN {X 0,Y 291.6,Z 301.782,A -85,B 0,C 180,E1 -16554.468,E2 -16554.468} C_VEL
LIN {X 0,Y 291.874,Z 301.751,A -85,B 0,C 180,E1 -16558.62,E2 -16558.62} C_VEL
LIN {X 0,Y 291.871,Z 301.751,A -85,B 0,C 180,E1 -16561.38,E2 -16561.38} C_VEL
LIN {X 0,Y 291.689,Z 301.778,A -85,B 0,C 180,E1 -16566.919,E2 -16566.919} C_VEL
LIN {X 0,Y 291.559,Z 301.784,A -85,B 0,C 180,E1 -16569.714,E2 -16569.714} C_VEL
LIN {X 0,Y 291.505,Z 301.79,A -85,B 0,C 180,E1 -16573.951,E2 -16573.951} C_VEL
LIN {X 0,Y 291.42,Z 301.807,A -85,B 0,C 180,E1 -16576.822,E2 -16576.822} C_VEL
LIN {X 0,Y 291.383,Z 301.817,A -85,B 0,C 180,E1 -16579.842,E2 -16579.842} C_VEL
LIN {X 0,Y 291.326,Z 301.825,A -85,B 0,C 180,E1 -16584.212,E2 -16584.212} C_VEL
LIN {X 0,Y 291.343,Z 301.819,A -85,B 0,C 180,E1 -16587.279,E2 -16587.279} C_VEL
LIN {X 0,Y 291.311,Z 301.823,A -85,B 0,C 180,E1 -16590.44,E2 -16590.44} C_VEL
LIN {X 0,Y 291.337,Z 301.812,A -85,B 0,C 180,E1 -16593.699,E2 -16593.699} C_VEL
LIN {X 0,Y 291.348,Z 301.815,A -85,B 0,C 180,E1 -16597.249,E2 -16597.249} C_VEL
LIN {X 0,Y 291.288,Z 301.804,A -85,B 0,C 180,E1 -16601.589,E2 -16601.589} C_VEL
LIN {X 0,Y 291.323,Z 301.967,A -85,B 0,C 180,E1 -16605.089,E2 -16605.089} C_VEL
LIN {X 0,Y 294.501,Z 312.224,A -85,B 0,C 180,E1 -16608.738,E2 -16608.738} C_VEL
LIN {X 0,Y 294.973,Z 313.788,A -85,B 0,C 180,E1 -16609.219,E2 -16609.219} C_VEL
LIN {X 0,Y 303.556,Z 329.262,A -85,B 0,C 180,E1 -16611.055,E2 -16611.055} C_VEL
LIN {X 0,Y 311.378,Z 344.915,A -85,B 0,C 180,E1 -16612.647,E2 -16612.647} C_VEL
LIN {X 0,Y 318.224,Z 360.68,A -85,B 0,C 180,E1 -16614.006,E2 -16614.006} C_VEL
LIN {X 0,Y 319.739,Z 370.881,A -85,B 0,C 180,E1 -16614.478,E2 -16614.478} C_VEL
LIN {X 0,Y 315.518,Z 480.329,A -85,B 0,C 180,E1 -16616.927,E2 -16616.927} C_VEL
LIN {X 0,Y 314.249,Z 495.738,A -85,B 0,C 180,E1 -16617.491,E2 -16617.491} C_VEL
LIN {X 0,Y 312.419,Z 510.64,A -85,B 0,C 180,E1 -16618.277,E2 -16618.277} C_VEL
LIN {X 0,Y 310.318,Z 524.851,A -85,B 0,C 180,E1 -16619.294,E2 -16619.294} C_VEL
LIN {X 0,Y 307.798,Z 539.08,A -85,B 0,C 180,E1 -16620.6,E2 -16620.6} C_VEL
LIN {X 0,Y 304.931,Z 552.804,A -85,B 0,C 180,E1 -16622.179,E2 -16622.179} C_VEL
LIN {X 0,Y 302.07,Z 565.234,A -85,B 0,C 180,E1 -16623.951,E2 -16623.951} C_VEL
LIN {X 0,Y 299.21,Z 577.43,A -85,B 0,C 180,E1 -16626.098,E2 -16626.098} C_VEL
LIN {X 0,Y 296.629,Z 588.285,A -85,B 0,C 180,E1 -16628.455,E2 -16628.455} C_VEL
LIN {X 0,Y 294.336,Z 597.327,A -85,B 0,C 180,E1 -16630.834,E2 -16630.834} C_VEL
LIN {X 0,Y 292.6,Z 604.835,A -85,B 0,C 180,E1 -16633.248,E2 -16633.248} C_VEL
LIN {X 0,Y 291.127,Z 611.845,A -85,B 0,C 180,E1 -16636.031,E2 -16636.031} C_VEL
LIN {X 0,Y 290.117,Z 617.361,A -85,B 0,C 180,E1 -16638.826,E2 -16638.826} C_VEL
LIN {X 0,Y 289.617,Z 621.538,A -85,B 0,C 180,E1 -16641.628,E2 -16641.628} C_VEL
LIN {X 0,Y 289.427,Z 624.619,A -85,B 0,C 180,E1 -16644.61,E2 -16644.61} C_VEL
LIN {X 0,Y 289.419,Z 626.219,A -85,B 0,C 180,E1 -16647.216,E2 -16647.216} C_VEL
LIN {X 0,Y 289.435,Z 626.817,A -85,B 0,C 180,E1 -16650,E2 -16650} C_VEL
LIN {X 0,Y 289.418,Z 626.208,A -85,B 0,C 180,E1 -16652.784,E2 -16652.784} C_VEL
LIN {X 0,Y 289.432,Z 624.446,A -85,B 0,C 180,E1 -16655.574,E2 -16655.574} C_VEL
LIN {X 0,Y 289.614,Z 621.506,A -85,B 0,C 180,E1 -16658.372,E2 -16658.372} C_VEL
LIN {X 0,Y 290.116,Z 617.324,A -85,B 0,C 180,E1 -16661.174,E2 -16661.174} C_VEL
LIN {X 0,Y 291.115,Z 611.791,A -85,B 0,C 180,E1 -16663.97,E2 -16663.97} C_VEL
LIN {X 0,Y 292.34,Z 605.825,A -85,B 0,C 180,E1 -16666.372,E2 -16666.372} C_VEL
LIN {X 0,Y 294.341,Z 597.243,A -85,B 0,C 180,E1 -16669.166,E2 -16669.166} C_VEL
LIN {X 0,Y 296.643,Z 588.191,A -85,B 0,C 180,E1 -16671.544,E2 -16671.544} C_VEL
LIN {X 0,Y 299.241,Z 577.312,A -85,B 0,C 180,E1 -16673.899,E2 -16673.899} C_VEL
LIN {X 0,Y 301.917,Z 566.116,A -85,B 0,C 180,E1 -16675.877,E2 -16675.877} C_VEL
LIN {X 0,Y 304.662,Z 553.853,A -85,B 0,C 180,E1 -16677.661,E2 -16677.661} C_VEL
LIN {X 0,Y 307.5,Z 540.374,A -85,B 0,C 180,E1 -16679.243,E2 -16679.243} C_VEL
LIN {X 0,Y 310.108,Z 525.546,A -85,B 0,C 180,E1 -16680.634,E2 -16680.634} C_VEL
LIN {X 0,Y 312.223,Z 511.515,A -85,B 0,C 180,E1 -16681.651,E2 -16681.651} C_VEL
LIN {X 0,Y 314.127,Z 496.098,A -85,B 0,C 180,E1 -16682.476,E2 -16682.476} C_VEL
LIN {X 0,Y 315.389,Z 480.854,A -85,B 0,C 180,E1 -16683.041,E2 -16683.041} C_VEL
LIN {X 0,Y 318.975,Z 389.083,A -85,B 0,C 180,E1 -16685.099,E2 -16685.099} C_VEL
LIN {X 0,Y 319.6,Z 369.458,A -85,B 0,C 180,E1 -16685.548,E2 -16685.548} C_VEL
LIN {X 0,Y 317.839,Z 359.694,A -85,B 0,C 180,E1 -16686.04,E2 -16686.04} C_VEL
LIN {X 0,Y 310.348,Z 342.758,A -85,B 0,C 180,E1 -16687.525,E2 -16687.525} C_VEL
LIN {X 0,Y 302.394,Z 327.035,A -85,B 0,C 180,E1 -16689.151,E2 -16689.151} C_VEL
LIN {X 0,Y 296.337,Z 316.442,A -85,B 0,C 180,E1 -16690.432,E2 -16690.432} C_VEL
LIN {X 0,Y 294.834,Z 313.42,A -85,B 0,C 180,E1 -16690.815,E2 -16690.815} C_VEL
LIN {X 0,Y 292.222,Z 304.814,A -85,B 0,C 180,E1 -16693.821,E2 -16693.821} C_VEL
LIN {X 0,Y 291.32,Z 301.822,A -85,B 0,C 180,E1 -16694.923,E2 -16694.923} C_VEL
LIN {X 0,Y 291.288,Z 301.823,A -85,B 0,C 180,E1 -16699.35,E2 -16699.35} C_VEL
LIN {X 0,Y 291.38,Z 301.814,A -85,B 0,C 180,E1 -16702.916,E2 -16702.916} C_VEL
LIN {X 0,Y 291.336,Z 301.817,A -85,B 0,C 180,E1 -16706.301,E2 -16706.301} C_VEL
LIN {X 0,Y 291.357,Z 301.812,A -85,B 0,C 180,E1 -16710.268,E2 -16710.268} C_VEL
LIN {X 0,Y 291.335,Z 301.821,A -85,B 0,C 180,E1 -16714.264,E2 -16714.264} C_VEL
LIN {X 0,Y 291.343,Z 301.818,A -85,B 0,C 180,E1 -16717.297,E2 -16717.297} C_VEL
LIN {X 0,Y 291.38,Z 301.787,A -85,B 0,C 180,E1 -16720.265,E2 -16720.265} C_VEL
LIN {X 0,Y 291.49,Z 301.8,A -85,B 0,C 180,E1 -16724.665,E2 -16724.665} C_VEL
LIN {X 0,Y 291.517,Z 301.76,A -85,B 0,C 180,E1 -16728.88,E2 -16728.88} C_VEL
LIN {X 0,Y 291.623,Z 301.782,A -85,B 0,C 180,E1 -16731.686,E2 -16731.686} C_VEL
LIN {X 0,Y 291.591,Z 301.778,A -85,B 0,C 180,E1 -16734.468,E2 -16734.468} C_VEL
LIN {X 0,Y 291.87,Z 301.743,A -85,B 0,C 180,E1 -16738.62,E2 -16738.62} C_VEL
LIN {X 0,Y 291.862,Z 301.752,A -85,B 0,C 180,E1 -16741.38,E2 -16741.38} C_VEL
LIN {X 0,Y 291.689,Z 301.768,A -85,B 0,C 180,E1 -16746.919,E2 -16746.919} C_VEL
LIN {X 0,Y 291.56,Z 301.789,A -85,B 0,C 180,E1 -16749.714,E2 -16749.714} C_VEL
LIN {X 0,Y 291.506,Z 301.795,A -85,B 0,C 180,E1 -16753.951,E2 -16753.951} C_VEL
LIN {X 0,Y 291.42,Z 301.81,A -85,B 0,C 180,E1 -16756.822,E2 -16756.822} C_VEL
LIN {X 0,Y 291.384,Z 301.784,A -85,B 0,C 180,E1 -16759.843,E2 -16759.843} C_VEL
LIN {X 0,Y 291.366,Z 301.816,A -85,B 0,C 180,E1 -16764.208,E2 -16764.208} C_VEL
LIN {X 0,Y 291.395,Z 301.785,A -85,B 0,C 180,E1 -16767.274,E2 -16767.274} C_VEL
LIN {X 0,Y 291.327,Z 301.821,A -85,B 0,C 180,E1 -16770.438,E2 -16770.438} C_VEL
LIN {X 0,Y 291.338,Z 301.819,A -85,B 0,C 180,E1 -16773.699,E2 -16773.699} C_VEL
LIN {X 0,Y 291.366,Z 301.811,A -85,B 0,C 180,E1 -16777.253,E2 -16777.253} C_VEL
LIN {X 0,Y 291.328,Z 301.817,A -85,B 0,C 180,E1 -16780.644,E2 -16780.644} C_VEL
LIN {X 0,Y 291.286,Z 301.824,A -85,B 0,C 180,E1 -16784.403,E2 -16784.403} C_VEL
LIN {X 0,Y 291.362,Z 301.828,A -85,B 0,C 180,E1 -16788.714,E2 -16788.714} C_VEL
LIN {X 0,Y 292.217,Z 304.459,A -85,B 0,C 180,E1 -16788.946,E2 -16788.946} C_VEL
LIN {X 0,Y 294.277,Z 307.039,A -85,B 0,C 180,E1 -16789.379,E2 -16789.379} C_VEL
LIN {X 0,Y 296.376,Z 310.333,A -85,B 0,C 180,E1 -16789.832,E2 -16789.832} C_VEL
LIN {X 0,Y 302.077,Z 319.475,A -85,B 0,C 180,E1 -16791.021,E2 -16791.021} C_VEL
LIN {X 0,Y 310.116,Z 334.362,A -85,B 0,C 180,E1 -16792.65,E2 -16792.65} C_VEL
LIN {X 0,Y 318.05,Z 350.981,A -85,B 0,C 180,E1 -16794.197,E2 -16794.197} C_VEL
LIN {X 0,Y 320.065,Z 355.552,A -85,B 0,C 180,E1 -16794.583,E2 -16794.583} C_VEL
LIN {X 0,Y 316.82,Z 444.121,A -85,B 0,C 180,E1 -16796.558,E2 -16796.558} C_VEL
LIN {X 0,Y 315.705,Z 468.072,A -85,B 0,C 180,E1 -16797.139,E2 -16797.139} C_VEL
LIN {X 0,Y 314.508,Z 482.736,A -85,B 0,C 180,E1 -16797.725,E2 -16797.725} C_VEL
LIN {X 0,Y 312.876,Z 497.334,A -85,B 0,C 180,E1 -16798.555,E2 -16798.555} C_VEL
LIN {X 0,Y 311.159,Z 510.242,A -85,B 0,C 180,E1 -16799.525,E2 -16799.525} C_VEL
LIN {X 0,Y 308.623,Z 524.647,A -85,B 0,C 180,E1 -16800.873,E2 -16800.873} C_VEL
LIN {X 0,Y 305.978,Z 538.097,A -85,B 0,C 180,E1 -16802.468,E2 -16802.468} C_VEL
LIN {X 0,Y 303.218,Z 550.303,A -85,B 0,C 180,E1 -16804.242,E2 -16804.242} C_VEL
LIN {X 0,Y 301.197,Z 559.199,A -85,B 0,C 180,E1 -16805.807,E2 -16805.807} C_VEL
LIN {X 0,Y 298.624,Z 569.285,A -85,B 0,C 180,E1 -16807.88,E2 -16807.88} C_VEL
LIN {X 0,Y 296.267,Z 578.724,A -85,B 0,C 180,E1 -16810.243,E2 -16810.243} C_VEL
LIN {X 0,Y 294.184,Z 586.584,A -85,B 0,C 180,E1 -16812.626,E2 -16812.626} C_VEL
LIN {X 0,Y 292.536,Z 593.906,A -85,B 0,C 180,E1 -16815.389,E2 -16815.389} C_VEL
LIN {X 0,Y 291.163,Z 599.719,A -85,B 0,C 180,E1 -16818.161,E2 -16818.161} C_VEL
LIN {X 0,Y 290.519,Z 603.156,A -85,B 0,C 180,E1 -16820.251,E2 -16820.251} C_VEL
LIN {X 0,Y 289.948,Z 606.636,A -85,B 0,C 180,E1 -16823.039,E2 -16823.039} C_VEL
LIN {X 0,Y 289.625,Z 608.935,A -85,B 0,C 180,E1 -16825.825,E2 -16825.825} C_VEL
LIN {X 0,Y 289.448,Z 610.108,A -85,B 0,C 180,E1 -16828.609,E2 -16828.609} C_VEL
LIN {X 0,Y 289.448,Z 610.122,A -85,B 0,C 180,E1 -16831.391,E2 -16831.391} C_VEL
LIN {X 0,Y 289.616,Z 609.003,A -85,B 0,C 180,E1 -16834.175,E2 -16834.175} C_VEL
LIN {X 0,Y 289.889,Z 606.759,A -85,B 0,C 180,E1 -16836.962,E2 -16836.962} C_VEL
LIN {X 0,Y 290.503,Z 603.326,A -85,B 0,C 180,E1 -16839.75,E2 -16839.75} C_VEL
LIN {X 0,Y 291.374,Z 598.629,A -85,B 0,C 180,E1 -16842.537,E2 -16842.537} C_VEL
LIN {X 0,Y 292.887,Z 592.531,A -85,B 0,C 180,E1 -16845.304,E2 -16845.304} C_VEL
LIN {X 0,Y 294.676,Z 584.857,A -85,B 0,C 180,E1 -16848.062,E2 -16848.062} C_VEL
LIN {X 0,Y 296.794,Z 576.666,A -85,B 0,C 180,E1 -16850.442,E2 -16850.442} C_VEL
LIN {X 0,Y 299.341,Z 566.794,A -85,B 0,C 180,E1 -16852.792,E2 -16852.792} C_VEL
LIN {X 0,Y 301.741,Z 556.673,A -85,B 0,C 180,E1 -16854.786,E2 -16854.786} C_VEL
LIN {X 0,Y 304.605,Z 544.611,A -85,B 0,C 180,E1 -16856.737,E2 -16856.737} C_VEL
LIN {X 0,Y 307.133,Z 532.516,A -85,B 0,C 180,E1 -16858.346,E2 -16858.346} C_VEL
LIN {X 0,Y 309.652,Z 519.365,A -85,B 0,C 180,E1 -16859.767,E2 -16859.767} C_VEL
LIN {X 0,Y 311.901,Z 505.12,A -85,B 0,C 180,E1 -16861,E2 -16861} C_VEL
LIN {X 0,Y 313.692,Z 490.857,A -85,B 0,C 180,E1 -16861.956,E2 -16861.956} C_VEL
LIN {X 0,Y 315.162,Z 475.958,A -85,B 0,C 180,E1 -16862.687,E2 -16862.687} C_VEL
LIN {X 0,Y 316.262,Z 460.615,A -85,B 0,C 180,E1 -16863.175,E2 -16863.175} C_VEL
LIN {X 0,Y 320.118,Z 355.606,A -85,B 0,C 180,E1 -16865.529,E2 -16865.529} C_VEL
LIN {X 0,Y 312.609,Z 339.3,A -85,B 0,C 180,E1 -16866.984,E2 -16866.984} C_VEL
LIN {X 0,Y 307.119,Z 328.545,A -85,B 0,C 180,E1 -16868.077,E2 -16868.077} C_VEL
LIN {X 0,Y 304.203,Z 324.383,A -85,B 0,C 180,E1 -16868.635,E2 -16868.635} C_VEL
LIN {X 0,Y 298.219,Z 319.009,A -85,B 0,C 180,E1 -16869.731,E2 -16869.731} C_VEL
LIN {X 0,Y 290.858,Z 312.908,A -85,B 0,C 180,E1 -16871.151,E2 -16871.151} C_VEL
LIN {X 0,Y 288.724,Z 310.432,A -85,B 0,C 180,E1 -16871.605,E2 -16871.605} C_VEL
LIN {X 0,Y 286.785,Z 307.291,A -85,B 0,C 180,E1 -16872.056,E2 -16872.056} C_VEL
LIN {X 0,Y 285.002,Z 305.057,A -85,B 0,C 180,E1 -16872.458,E2 -16872.458} C_VEL
LIN {X 0,Y 284.275,Z 302.7,A -85,B 0,C 180,E1 -16872.696,E2 -16872.696} C_VEL
LIN {X 0,Y 284.253,Z 302.703,A -85,B 0,C 180,E1 -16876.188,E2 -16876.188} C_VEL
LIN {X 0,Y 284.302,Z 302.693,A -85,B 0,C 180,E1 -16880.023,E2 -16880.023} C_VEL
LIN {X 0,Y 284.317,Z 302.67,A -85,B 0,C 180,E1 -16883.612,E2 -16883.612} C_VEL
LIN {X 0,Y 284.3,Z 302.689,A -85,B 0,C 180,E1 -16887.19,E2 -16887.19} C_VEL
LIN {X 0,Y 284.338,Z 302.666,A -85,B 0,C 180,E1 -16890.374,E2 -16890.374} C_VEL
LIN {X 0,Y 284.347,Z 302.687,A -85,B 0,C 180,E1 -16893.583,E2 -16893.583} C_VEL
LIN {X 0,Y 284.323,Z 302.695,A -85,B 0,C 180,E1 -16896.703,E2 -16896.703} C_VEL
LIN {X 0,Y 284.37,Z 302.687,A -85,B 0,C 180,E1 -16899.904,E2 -16899.904} C_VEL
LIN {X 0,Y 284.439,Z 302.68,A -85,B 0,C 180,E1 -16904.492,E2 -16904.492} C_VEL
LIN {X 0,Y 284.473,Z 302.675,A -85,B 0,C 180,E1 -16908.601,E2 -16908.601} C_VEL
LIN {X 0,Y 284.612,Z 302.648,A -85,B 0,C 180,E1 -16911.48,E2 -16911.48} C_VEL
LIN {X 0,Y 284.57,Z 302.659,A -85,B 0,C 180,E1 -16914.33,E2 -16914.33} C_VEL
LIN {X 0,Y 284.84,Z 302.627,A -85,B 0,C 180,E1 -16918.586,E2 -16918.586} C_VEL
LIN {X 0,Y 284.837,Z 302.627,A -85,B 0,C 180,E1 -16921.414,E2 -16921.414} C_VEL
LIN {X 0,Y 284.643,Z 302.654,A -85,B 0,C 180,E1 -16927.091,E2 -16927.091} C_VEL
LIN {X 0,Y 284.505,Z 302.664,A -85,B 0,C 180,E1 -16929.957,E2 -16929.957} C_VEL
LIN {X 0,Y 284.454,Z 302.67,A -85,B 0,C 180,E1 -16934.304,E2 -16934.304} C_VEL
LIN {X 0,Y 284.323,Z 302.69,A -85,B 0,C 180,E1 -16938.744,E2 -16938.744} C_VEL
LIN {X 0,Y 284.302,Z 302.697,A -85,B 0,C 180,E1 -16943.298,E2 -16943.298} C_VEL
LIN {X 0,Y 284.319,Z 302.694,A -85,B 0,C 180,E1 -16947.146,E2 -16947.146} C_VEL
LIN {X 0,Y 284.289,Z 302.699,A -85,B 0,C 180,E1 -16950.092,E2 -16950.092} C_VEL
LIN {X 0,Y 284.298,Z 302.687,A -85,B 0,C 180,E1 -16952.946,E2 -16952.946} C_VEL
LIN {X 0,Y 284.312,Z 302.688,A -85,B 0,C 180,E1 -16956.389,E2 -16956.389} C_VEL
LIN {X 0,Y 284.249,Z 302.677,A -85,B 0,C 180,E1 -16960.004,E2 -16960.004} C_VEL
LIN {X 0,Y 284.245,Z 302.796,A -85,B 0,C 180,E1 -16964.007,E2 -16964.007} C_VEL
LIN {X 0,Y 287.67,Z 313.524,A -85,B 0,C 180,E1 -16967.951,E2 -16967.951} C_VEL
LIN {X 0,Y 296.163,Z 328.524,A -85,B 0,C 180,E1 -16969.874,E2 -16969.874} C_VEL
LIN {X 0,Y 304.148,Z 344.041,A -85,B 0,C 180,E1 -16971.581,E2 -16971.581} C_VEL
LIN {X 0,Y 311.765,Z 361.02,A -85,B 0,C 180,E1 -16973.155,E2 -16973.155} C_VEL
LIN {X 0,Y 312.829,Z 364.021,A -85,B 0,C 180,E1 -16973.384,E2 -16973.384} C_VEL
LIN {X 0,Y 313.952,Z 371.99,A -85,B 0,C 180,E1 -16973.756,E2 -16973.756} C_VEL
LIN {X 0,Y 309.584,Z 480.142,A -85,B 0,C 180,E1 -16976.209,E2 -16976.209} C_VEL
LIN {X 0,Y 308.29,Z 495.545,A -85,B 0,C 180,E1 -16976.783,E2 -16976.783} C_VEL
LIN {X 0,Y 306.395,Z 510.445,A -85,B 0,C 180,E1 -16977.578,E2 -16977.578} C_VEL
LIN {X 0,Y 304.135,Z 525.111,A -85,B 0,C 180,E1 -16978.644,E2 -16978.644} C_VEL
LIN {X 0,Y 301.598,Z 538.88,A -85,B 0,C 180,E1 -16979.934,E2 -16979.934} C_VEL
LIN {X 0,Y 298.658,Z 552.605,A -85,B 0,C 180,E1 -16981.542,E2 -16981.542} C_VEL
LIN {X 0,Y 295.686,Z 565.034,A -85,B 0,C 180,E1 -16983.345,E2 -16983.345} C_VEL
LIN {X 0,Y 292.686,Z 577.228,A -85,B 0,C 180,E1 -16985.531,E2 -16985.531} C_VEL
LIN {X 0,Y 290.354,Z 586.643,A -85,B 0,C 180,E1 -16987.591,E2 -16987.591} C_VEL
LIN {X 0,Y 287.851,Z 595.903,A -85,B 0,C 180,E1 -16990.013,E2 -16990.013} C_VEL
LIN {X 0,Y 285.713,Z 604.631,A -85,B 0,C 180,E1 -16992.832,E2 -16992.832} C_VEL
LIN {X 0,Y 284.174,Z 611.641,A -85,B 0,C 180,E1 -16995.682,E2 -16995.682} C_VEL
LIN {X 0,Y 283.096,Z 617.157,A -85,B 0,C 180,E1 -16998.545,E2 -16998.545} C_VEL
LIN {X 0,Y 282.557,Z 621.334,A -85,B 0,C 180,E1 -17001.418,E2 -17001.418} C_VEL
LIN {X 0,Y 282.339,Z 624.266,A -85,B 0,C 180,E1 -17004.286,E2 -17004.286} C_VEL
LIN {X 0,Y 282.325,Z 626.016,A -85,B 0,C 180,E1 -17007.146,E2 -17007.146} C_VEL
LIN {X 0,Y 282.354,Z 626.614,A -85,B 0,C 180,E1 -17010,E2 -17010} C_VEL
LIN {X 0,Y 282.324,Z 626.005,A -85,B 0,C 180,E1 -17012.854,E2 -17012.854} C_VEL
LIN {X 0,Y 282.335,Z 624.242,A -85,B 0,C 180,E1 -17015.714,E2 -17015.714} C_VEL
LIN {X 0,Y 282.553,Z 621.301,A -85,B 0,C 180,E1 -17018.583,E2 -17018.583} C_VEL
LIN {X 0,Y 283.095,Z 617.118,A -85,B 0,C 180,E1 -17021.455,E2 -17021.455} C_VEL
LIN {X 0,Y 284.157,Z 611.585,A -85,B 0,C 180,E1 -17024.319,E2 -17024.319} C_VEL
LIN {X 0,Y 285.249,Z 606.44,A -85,B 0,C 180,E1 -17026.459,E2 -17026.459} C_VEL
LIN {X 0,Y 287.009,Z 599.289,A -85,B 0,C 180,E1 -17028.932,E2 -17028.932} C_VEL
LIN {X 0,Y 289.269,Z 590.707,A -85,B 0,C 180,E1 -17031.372,E2 -17031.372} C_VEL
LIN {X 0,Y 291.85,Z 580.395,A -85,B 0,C 180,E1 -17033.784,E2 -17033.784} C_VEL
LIN {X 0,Y 294.471,Z 569.826,A -85,B 0,C 180,E1 -17035.82,E2 -17035.82} C_VEL
LIN {X 0,Y 297.283,Z 558.357,A -85,B 0,C 180,E1 -17037.641,E2 -17037.641} C_VEL
LIN {X 0,Y 300.104,Z 545.89,A -85,B 0,C 180,E1 -17039.265,E2 -17039.265} C_VEL
LIN {X 0,Y 302.808,Z 532.234,A -85,B 0,C 180,E1 -17040.703,E2 -17040.703} C_VEL
LIN {X 0,Y 305.197,Z 518.088,A -85,B 0,C 180,E1 -17041.883,E2 -17041.883} C_VEL
LIN {X 0,Y 307.284,Z 503.522,A -85,B 0,C 180,E1 -17042.803,E2 -17042.803} C_VEL
LIN {X 0,Y 308.894,Z 488.568,A -85,B 0,C 180,E1 -17043.485,E2 -17043.485} C_VEL
LIN {X 0,Y 309.876,Z 473.175,A -85,B 0,C 180,E1 -17043.951,E2 -17043.951} C_VEL
LIN {X 0,Y 313.846,Z 371.687,A -85,B 0,C 180,E1 -17046.234,E2 -17046.234} C_VEL
LIN {X 0,Y 312.424,Z 362.711,A -85,B 0,C 180,E1 -17046.675,E2 -17046.675} C_VEL
LIN {X 0,Y 304.162,Z 344.098,A -85,B 0,C 180,E1 -17048.379,E2 -17048.379} C_VEL
LIN {X 0,Y 297.225,Z 330.578,A -85,B 0,C 180,E1 -17049.852,E2 -17049.852} C_VEL
LIN {X 0,Y 291.943,Z 321.148,A -85,B 0,C 180,E1 -17051.015,E2 -17051.015} C_VEL
LIN {X 0,Y 287.542,Z 313.305,A -85,B 0,C 180,E1 -17052.035,E2 -17052.035} C_VEL
LIN {X 0,Y 284.839,Z 304.772,A -85,B 0,C 180,E1 -17055.186,E2 -17055.186} C_VEL
LIN {X 0,Y 284.243,Z 302.707,A -85,B 0,C 180,E1 -17056.057,E2 -17056.057} C_VEL
LIN {X 0,Y 284.25,Z 302.7,A -85,B 0,C 180,E1 -17060.036,E2 -17060.036} C_VEL
LIN {X 0,Y 284.312,Z 302.693,A -85,B 0,C 180,E1 -17063.611,E2 -17063.611} C_VEL
LIN {X 0,Y 284.299,Z 302.69,A -85,B 0,C 180,E1 -17067.19,E2 -17067.19} C_VEL
LIN {X 0,Y 284.329,Z 302.688,A -85,B 0,C 180,E1 -17070.373,E2 -17070.373} C_VEL
LIN {X 0,Y 284.29,Z 302.693,A -85,B 0,C 180,E1 -17073.578,E2 -17073.578} C_VEL
LIN {X 0,Y 284.3,Z 302.693,A -85,B 0,C 180,E1 -17076.701,E2 -17076.701} C_VEL
LIN {X 0,Y 284.323,Z 302.662,A -85,B 0,C 180,E1 -17081.256,E2 -17081.256} C_VEL
LIN {X 0,Y 284.454,Z 302.671,A -85,B 0,C 180,E1 -17085.696,E2 -17085.696} C_VEL
LIN {X 0,Y 284.502,Z 302.645,A -85,B 0,C 180,E1 -17090.043,E2 -17090.043} C_VEL
LIN {X 0,Y 284.631,Z 302.656,A -85,B 0,C 180,E1 -17092.908,E2 -17092.908} C_VEL
LIN {X 0,Y 284.836,Z 302.619,A -85,B 0,C 180,E1 -17098.586,E2 -17098.586} C_VEL
LIN {X 0,Y 284.829,Z 302.627,A -85,B 0,C 180,E1 -17101.414,E2 -17101.414} C_VEL
LIN {X 0,Y 284.644,Z 302.645,A -85,B 0,C 180,E1 -17107.092,E2 -17107.092} C_VEL
LIN {X 0,Y 284.506,Z 302.666,A -85,B 0,C 180,E1 -17109.958,E2 -17109.958} C_VEL
LIN {X 0,Y 284.455,Z 302.672,A -85,B 0,C 180,E1 -17114.304,E2 -17114.304} C_VEL
LIN {X 0,Y 284.325,Z 302.676,A -85,B 0,C 180,E1 -17118.744,E2 -17118.744} C_VEL
LIN {X 0,Y 284.324,Z 302.689,A -85,B 0,C 180,E1 -17123.297,E2 -17123.297} C_VEL
LIN {X 0,Y 284.372,Z 302.66,A -85,B 0,C 180,E1 -17127.167,E2 -17127.167} C_VEL
LIN {X 0,Y 284.305,Z 302.695,A -85,B 0,C 180,E1 -17130.098,E2 -17130.098} C_VEL
LIN {X 0,Y 284.3,Z 302.694,A -85,B 0,C 180,E1 -17132.946,E2 -17132.946} C_VEL
LIN {X 0,Y 284.325,Z 302.693,A -85,B 0,C 180,E1 -17136.387,E2 -17136.387} C_VEL
LIN {X 0,Y 284.301,Z 302.69,A -85,B 0,C 180,E1 -17139.996,E2 -17139.996} C_VEL
LIN {X 0,Y 284.242,Z 302.702,A -85,B 0,C 180,E1 -17144.191,E2 -17144.191} C_VEL
LIN {X 0,Y 284.29,Z 302.765,A -85,B 0,C 180,E1 -17147.471,E2 -17147.471} C_VEL
LIN {X 0,Y 285.216,Z 305.462,A -85,B 0,C 180,E1 -17147.733,E2 -17147.733} C_VEL
LIN {X 0,Y 287.306,Z 307.973,A -85,B 0,C 180,E1 -17148.197,E2 -17148.197} C_VEL
LIN {X 0,Y 289.483,Z 311.359,A -85,B 0,C 180,E1 -17148.694,E2 -17148.694} C_VEL
LIN {X 0,Y 296.868,Z 322.809,A -85,B 0,C 180,E1 -17150.299,E2 -17150.299} C_VEL
LIN {X 0,Y 305.224,Z 338.431,A -85,B 0,C 180,E1 -17152.059,E2 -17152.059} C_VEL
LIN {X 0,Y 313.084,Z 355.088,A -85,B 0,C 180,E1 -17153.648,E2 -17153.648} C_VEL
LIN {X 0,Y 314.277,Z 357.823,A -85,B 0,C 180,E1 -17153.886,E2 -17153.886} C_VEL
LIN {X 0,Y 310.113,Z 463.086,A -85,B 0,C 180,E1 -17156.274,E2 -17156.274} C_VEL
LIN {X 0,Y 308.94,Z 478.464,A -85,B 0,C 180,E1 -17156.813,E2 -17156.813} C_VEL
LIN {X 0,Y 307.408,Z 493.075,A -85,B 0,C 180,E1 -17157.581,E2 -17157.581} C_VEL
LIN {X 0,Y 305.505,Z 507.333,A -85,B 0,C 180,E1 -17158.595,E2 -17158.595} C_VEL
LIN {X 0,Y 303.078,Z 521.722,A -85,B 0,C 180,E1 -17159.905,E2 -17159.905} C_VEL
LIN {X 0,Y 300.46,Z 534.487,A -85,B 0,C 180,E1 -17161.347,E2 -17161.347} C_VEL
LIN {X 0,Y 297.846,Z 546.279,A -85,B 0,C 180,E1 -17162.986,E2 -17162.986} C_VEL
LIN {X 0,Y 295.135,Z 557.202,A -85,B 0,C 180,E1 -17164.809,E2 -17164.809} C_VEL
LIN {X 0,Y 292.872,Z 566.489,A -85,B 0,C 180,E1 -17166.676,E2 -17166.676} C_VEL
LIN {X 0,Y 290.217,Z 576.445,A -85,B 0,C 180,E1 -17169.073,E2 -17169.073} C_VEL
LIN {X 0,Y 287.962,Z 584.699,A -85,B 0,C 180,E1 -17171.502,E2 -17171.502} C_VEL
LIN {X 0,Y 286.013,Z 592.445,A -85,B 0,C 180,E1 -17174.319,E2 -17174.319} C_VEL
LIN {X 0,Y 284.445,Z 598.609,A -85,B 0,C 180,E1 -17177.152,E2 -17177.152} C_VEL
LIN {X 0,Y 283.488,Z 603.361,A -85,B 0,C 180,E1 -17180.007,E2 -17180.007} C_VEL
LIN {X 0,Y 282.892,Z 606.84,A -85,B 0,C 180,E1 -17182.865,E2 -17182.865} C_VEL
LIN {X 0,Y 282.547,Z 609.138,A -85,B 0,C 180,E1 -17185.721,E2 -17185.721} C_VEL
LIN {X 0,Y 282.372,Z 610.311,A -85,B 0,C 180,E1 -17188.574,E2 -17188.574} C_VEL
LIN {X 0,Y 282.371,Z 610.324,A -85,B 0,C 180,E1 -17191.426,E2 -17191.426} C_VEL
LIN {X 0,Y 282.538,Z 609.206,A -85,B 0,C 180,E1 -17194.279,E2 -17194.279} C_VEL
LIN {X 0,Y 282.834,Z 606.961,A -85,B 0,C 180,E1 -17197.137,E2 -17197.137} C_VEL
LIN {X 0,Y 283.468,Z 603.53,A -85,B 0,C 180,E1 -17199.994,E2 -17199.994} C_VEL
LIN {X 0,Y 284.413,Z 598.831,A -85,B 0,C 180,E1 -17202.849,E2 -17202.849} C_VEL
LIN {X 0,Y 285.988,Z 592.734,A -85,B 0,C 180,E1 -17205.683,E2 -17205.683} C_VEL
LIN {X 0,Y 287.902,Z 585.059,A -85,B 0,C 180,E1 -17208.502,E2 -17208.502} C_VEL
LIN {X 0,Y 290.129,Z 576.867,A -85,B 0,C 180,E1 -17210.934,E2 -17210.934} C_VEL
LIN {X 0,Y 292.802,Z 566.994,A -85,B 0,C 180,E1 -17213.33,E2 -17213.33} C_VEL
LIN {X 0,Y 295.286,Z 556.874,A -85,B 0,C 180,E1 -17215.366,E2 -17215.366} C_VEL
LIN {X 0,Y 298.284,Z 544.81,A -85,B 0,C 180,E1 -17217.351,E2 -17217.351} C_VEL
LIN {X 0,Y 300.886,Z 532.715,A -85,B 0,C 180,E1 -17218.99,E2 -17218.99} C_VEL
LIN {X 0,Y 303.517,Z 519.562,A -85,B 0,C 180,E1 -17220.431,E2 -17220.431} C_VEL
LIN {X 0,Y 305.639,Z 506.784,A -85,B 0,C 180,E1 -17221.564,E2 -17221.564} C_VEL
LIN {X 0,Y 307.609,Z 491.822,A -85,B 0,C 180,E1 -17222.608,E2 -17222.608} C_VEL
LIN {X 0,Y 309.156,Z 477.061,A -85,B 0,C 180,E1 -17223.356,E2 -17223.356} C_VEL
LIN {X 0,Y 310.238,Z 462.301,A -85,B 0,C 180,E1 -17223.857,E2 -17223.857} C_VEL
LIN {X 0,Y 314.358,Z 357.828,A -85,B 0,C 180,E1 -17226.226,E2 -17226.226} C_VEL
LIN {X 0,Y 307.005,Z 341.995,A -85,B 0,C 180,E1 -17227.702,E2 -17227.702} C_VEL
LIN {X 0,Y 299.538,Z 327.522,A -85,B 0,C 180,E1 -17229.261,E2 -17229.261} C_VEL
LIN {X 0,Y 294.064,Z 318.363,A -85,B 0,C 180,E1 -17230.432,E2 -17230.432} C_VEL
LIN {X 0,Y 289.089,Z 310.895,A -85,B 0,C 180,E1 -17231.526,E2 -17231.526} C_VEL
LIN {X 0,Y 288.724,Z 310.432,A -85,B 0,C 180,E1 -17231.605,E2 -17231.605} C_VEL
LIN {X 0,Y 285.53,Z 307.311,A -85,B 0,C 180,E1 -17232.285,E2 -17232.285} C_VEL
LIN {X 0,Y 280.993,Z 304.859,A -85,B 0,C 180,E1 -17233.246,E2 -17233.246} C_VEL
LIN {X 0,Y 278.091,Z 303.835,A -85,B 0,C 180,E1 -17234.16,E2 -17234.16} C_VEL
LIN {X 0,Y 277.226,Z 303.587,A -85,B 0,C 180,E1 -17234.818,E2 -17234.818} C_VEL
LIN {X 0,Y 277.196,Z 303.579,A -85,B 0,C 180,E1 -17234.955,E2 -17234.955} C_VEL
LIN {X 0,Y 277.205,Z 303.561,A -85,B 0,C 180,E1 -17238.762,E2 -17238.762} C_VEL
LIN {X 0,Y 277.253,Z 303.552,A -85,B 0,C 180,E1 -17242.528,E2 -17242.528} C_VEL
LIN {X 0,Y 277.24,Z 303.576,A -85,B 0,C 180,E1 -17246.103,E2 -17246.103} C_VEL
LIN {X 0,Y 277.257,Z 303.542,A -85,B 0,C 180,E1 -17249.538,E2 -17249.538} C_VEL
LIN {X 0,Y 277.332,Z 303.566,A -85,B 0,C 180,E1 -17252.861,E2 -17252.861} C_VEL
LIN {X 0,Y 277.284,Z 303.57,A -85,B 0,C 180,E1 -17256.075,E2 -17256.075} C_VEL
LIN {X 0,Y 277.31,Z 303.567,A -85,B 0,C 180,E1 -17260.763,E2 -17260.763} C_VEL
LIN {X 0,Y 277.401,Z 303.552,A -85,B 0,C 180,E1 -17265.324,E2 -17265.324} C_VEL
LIN {X 0,Y 277.449,Z 303.547,A -85,B 0,C 180,E1 -17269.786,E2 -17269.786} C_VEL
LIN {X 0,Y 277.607,Z 303.529,A -85,B 0,C 180,E1 -17272.728,E2 -17272.728} C_VEL
LIN {X 0,Y 277.806,Z 303.503,A -85,B 0,C 180,E1 -17278.55,E2 -17278.55} C_VEL
LIN {X 0,Y 277.803,Z 303.503,A -85,B 0,C 180,E1 -17281.449,E2 -17281.449} C_VEL
LIN {X 0,Y 277.601,Z 303.531,A -85,B 0,C 180,E1 -17287.272,E2 -17287.272} C_VEL
LIN {X 0,Y 277.449,Z 303.544,A -85,B 0,C 180,E1 -17290.213,E2 -17290.213} C_VEL
LIN {X 0,Y 277.401,Z 303.552,A -85,B 0,C 180,E1 -17294.676,E2 -17294.676} C_VEL
LIN {X 0,Y 277.276,Z 303.573,A -85,B 0,C 180,E1 -17299.239,E2 -17299.239} C_VEL
LIN {X 0,Y 277.253,Z 303.577,A -85,B 0,C 180,E1 -17303.927,E2 -17303.927} C_VEL
LIN {X 0,Y 277.26,Z 303.574,A -85,B 0,C 180,E1 -17307.482,E2 -17307.482} C_VEL
LIN {X 0,Y 277.242,Z 303.575,A -85,B 0,C 180,E1 -17310.473,E2 -17310.473} C_VEL
LIN {X 0,Y 277.239,Z 303.569,A -85,B 0,C 180,E1 -17313.897,E2 -17313.897} C_VEL
LIN {X 0,Y 277.241,Z 303.574,A -85,B 0,C 180,E1 -17317.473,E2 -17317.473} C_VEL
LIN {X 0,Y 277.171,Z 303.558,A -85,B 0,C 180,E1 -17321.243,E2 -17321.243} C_VEL
LIN {X 0,Y 277.173,Z 303.684,A -85,B 0,C 180,E1 -17322.874,E2 -17322.874} C_VEL
LIN {X 0,Y 280.304,Z 313.289,A -85,B 0,C 180,E1 -17326.579,E2 -17326.579} C_VEL
LIN {X 0,Y 283.175,Z 318.004,A -85,B 0,C 180,E1 -17327.282,E2 -17327.282} C_VEL
LIN {X 0,Y 291.891,Z 333.532,A -85,B 0,C 180,E1 -17329.327,E2 -17329.327} C_VEL
LIN {X 0,Y 299.215,Z 347.861,A -85,B 0,C 180,E1 -17330.948,E2 -17330.948} C_VEL
LIN {X 0,Y 306.911,Z 365.361,A -85,B 0,C 180,E1 -17332.602,E2 -17332.602} C_VEL
LIN {X 0,Y 307.787,Z 369.652,A -85,B 0,C 180,E1 -17332.849,E2 -17332.849} C_VEL
LIN {X 0,Y 308.203,Z 372.689,A -85,B 0,C 180,E1 -17332.994,E2 -17332.994} C_VEL
LIN {X 0,Y 303.856,Z 476.952,A -85,B 0,C 180,E1 -17335.382,E2 -17335.382} C_VEL
LIN {X 0,Y 302.622,Z 492.607,A -85,B 0,C 180,E1 -17335.927,E2 -17335.927} C_VEL
LIN {X 0,Y 300.772,Z 507.644,A -85,B 0,C 180,E1 -17336.695,E2 -17336.695} C_VEL
LIN {X 0,Y 298.633,Z 521.626,A -85,B 0,C 180,E1 -17337.67,E2 -17337.67} C_VEL
LIN {X 0,Y 296.278,Z 534.617,A -85,B 0,C 180,E1 -17338.829,E2 -17338.829} C_VEL
LIN {X 0,Y 293.597,Z 547.226,A -85,B 0,C 180,E1 -17340.219,E2 -17340.219} C_VEL
LIN {X 0,Y 290.729,Z 559.467,A -85,B 0,C 180,E1 -17341.876,E2 -17341.876} C_VEL
LIN {X 0,Y 287.558,Z 571.676,A -85,B 0,C 180,E1 -17343.902,E2 -17343.902} C_VEL
LIN {X 0,Y 284.626,Z 582.695,A -85,B 0,C 180,E1 -17346.15,E2 -17346.15} C_VEL
LIN {X 0,Y 282.209,Z 591.963,A -85,B 0,C 180,E1 -17348.45,E2 -17348.45} C_VEL
LIN {X 0,Y 279.92,Z 600.295,A -85,B 0,C 180,E1 -17350.951,E2 -17350.951} C_VEL
LIN {X 0,Y 277.976,Z 608.227,A -85,B 0,C 180,E1 -17353.892,E2 -17353.892} C_VEL
LIN {X 0,Y 276.647,Z 614.373,A -85,B 0,C 180,E1 -17356.783,E2 -17356.783} C_VEL
LIN {X 0,Y 275.75,Z 619.203,A -85,B 0,C 180,E1 -17359.723,E2 -17359.723} C_VEL
LIN {X 0,Y 275.359,Z 622.749,A -85,B 0,C 180,E1 -17362.668,E2 -17362.668} C_VEL
LIN {X 0,Y 275.203,Z 625.082,A -85,B 0,C 180,E1 -17365.606,E2 -17365.606} C_VEL
LIN {X 0,Y 275.257,Z 626.257,A -85,B 0,C 180,E1 -17368.537,E2 -17368.537} C_VEL
LIN {X 0,Y 275.257,Z 626.254,A -85,B 0,C 180,E1 -17371.463,E2 -17371.463} C_VEL
LIN {X 0,Y 275.201,Z 625.064,A -85,B 0,C 180,E1 -17374.394,E2 -17374.394} C_VEL
LIN {X 0,Y 275.301,Z 622.716,A -85,B 0,C 180,E1 -17377.333,E2 -17377.333} C_VEL
LIN {X 0,Y 275.737,Z 619.166,A -85,B 0,C 180,E1 -17380.277,E2 -17380.277} C_VEL
LIN {X 0,Y 276.643,Z 614.325,A -85,B 0,C 180,E1 -17383.217,E2 -17383.217} C_VEL
LIN {X 0,Y 277.881,Z 608.058,A -85,B 0,C 180,E1 -17386.153,E2 -17386.153} C_VEL
LIN {X 0,Y 279.937,Z 600.206,A -85,B 0,C 180,E1 -17389.048,E2 -17389.048} C_VEL
LIN {X 0,Y 282.224,Z 591.862,A -85,B 0,C 180,E1 -17391.549,E2 -17391.549} C_VEL
LIN {X 0,Y 284.783,Z 582.248,A -85,B 0,C 180,E1 -17393.922,E2 -17393.922} C_VEL
LIN {X 0,Y 287.553,Z 571.539,A -85,B 0,C 180,E1 -17396.099,E2 -17396.099} C_VEL
LIN {X 0,Y 290.702,Z 559.304,A -85,B 0,C 180,E1 -17398.126,E2 -17398.126} C_VEL
LIN {X 0,Y 293.595,Z 547.027,A -85,B 0,C 180,E1 -17399.781,E2 -17399.781} C_VEL
LIN {X 0,Y 296.448,Z 533.293,A -85,B 0,C 180,E1 -17401.284,E2 -17401.284} C_VEL
LIN {X 0,Y 299.013,Z 518.915,A -85,B 0,C 180,E1 -17402.523,E2 -17402.523} C_VEL
LIN {X 0,Y 301.131,Z 504.633,A -85,B 0,C 180,E1 -17403.46,E2 -17403.46} C_VEL
LIN {X 0,Y 302.902,Z 489.275,A -85,B 0,C 180,E1 -17404.188,E2 -17404.188} C_VEL
LIN {X 0,Y 303.934,Z 474.462,A -85,B 0,C 180,E1 -17404.658,E2 -17404.658} C_VEL
LIN {X 0,Y 308.1,Z 372.886,A -85,B 0,C 180,E1 -17406.981,E2 -17406.981} C_VEL
LIN {X 0,Y 306.916,Z 365.514,A -85,B 0,C 180,E1 -17407.358,E2 -17407.358} C_VEL
LIN {X 0,Y 299.316,Z 348.163,A -85,B 0,C 180,E1 -17408.989,E2 -17408.989} C_VEL
LIN {X 0,Y 292.193,Z 334.151,A -85,B 0,C 180,E1 -17410.561,E2 -17410.561} C_VEL
LIN {X 0,Y 285.759,Z 322.561,A -85,B 0,C 180,E1 -17412.047,E2 -17412.047} C_VEL
LIN {X 0,Y 282.111,Z 316.578,A -85,B 0,C 180,E1 -17412.916,E2 -17412.916} C_VEL
LIN {X 0,Y 280.133,Z 312.913,A -85,B 0,C 180,E1 -17413.449,E2 -17413.449} C_VEL
LIN {X 0,Y 277.174,Z 303.582,A -85,B 0,C 180,E1 -17417.126,E2 -17417.126} C_VEL
LIN {X 0,Y 277.184,Z 303.584,A -85,B 0,C 180,E1 -17420.664,E2 -17420.664} C_VEL
LIN {X 0,Y 277.27,Z 303.566,A -85,B 0,C 180,E1 -17424.34,E2 -17424.34} C_VEL
LIN {X 0,Y 277.233,Z 303.572,A -85,B 0,C 180,E1 -17427.835,E2 -17427.835} C_VEL
LIN {X 0,Y 277.228,Z 303.576,A -85,B 0,C 180,E1 -17431.206,E2 -17431.206} C_VEL
LIN {X 0,Y 277.225,Z 303.578,A -85,B 0,C 180,E1 -17434.471,E2 -17434.471} C_VEL
LIN {X 0,Y 277.241,Z 303.578,A -85,B 0,C 180,E1 -17437.651,E2 -17437.651} C_VEL
LIN {X 0,Y 277.276,Z 303.539,A -85,B 0,C 180,E1 -17440.761,E2 -17440.761} C_VEL
LIN {X 0,Y 277.4,Z 303.554,A -85,B 0,C 180,E1 -17445.324,E2 -17445.324} C_VEL
LIN {X 0,Y 277.444,Z 303.519,A -85,B 0,C 180,E1 -17449.787,E2 -17449.787} C_VEL
LIN {X 0,Y 277.586,Z 303.533,A -85,B 0,C 180,E1 -17452.727,E2 -17452.727} C_VEL
LIN {X 0,Y 277.802,Z 303.495,A -85,B 0,C 180,E1 -17458.551,E2 -17458.551} C_VEL
LIN {X 0,Y 277.796,Z 303.503,A -85,B 0,C 180,E1 -17461.45,E2 -17461.45} C_VEL
LIN {X 0,Y 277.602,Z 303.523,A -85,B 0,C 180,E1 -17467.272,E2 -17467.272} C_VEL
LIN {X 0,Y 277.447,Z 303.545,A -85,B 0,C 180,E1 -17470.214,E2 -17470.214} C_VEL
LIN {X 0,Y 277.401,Z 303.548,A -85,B 0,C 180,E1 -17474.676,E2 -17474.676} C_VEL
LIN {X 0,Y 277.278,Z 303.546,A -85,B 0,C 180,E1 -17479.239,E2 -17479.239} C_VEL
LIN {X 0,Y 277.284,Z 303.57,A -85,B 0,C 180,E1 -17483.925,E2 -17483.925} C_VEL
LIN {X 0,Y 277.303,Z 303.539,A -85,B 0,C 180,E1 -17487.499,E2 -17487.499} C_VEL
LIN {X 0,Y 277.267,Z 303.573,A -85,B 0,C 180,E1 -17490.482,E2 -17490.482} C_VEL
LIN {X 0,Y 277.241,Z 303.575,A -85,B 0,C 180,E1 -17493.897,E2 -17493.897} C_VEL
LIN {X 0,Y 277.259,Z 303.567,A -85,B 0,C 180,E1 -17497.471,E2 -17497.471} C_VEL
LIN {X 0,Y 277.205,Z 303.581,A -85,B 0,C 180,E1 -17501.238,E2 -17501.238} C_VEL
LIN {X 0,Y 277.198,Z 303.58,A -85,B 0,C 180,E1 -17505.227,E2 -17505.227} C_VEL
LIN {X 0,Y 277.22,Z 303.61,A -85,B 0,C 180,E1 -17506.135,E2 -17506.135} C_VEL
LIN {X 0,Y 278.106,Z 306.25,A -85,B 0,C 180,E1 -17506.404,E2 -17506.404} C_VEL
LIN {X 0,Y 280.333,Z 308.96,A -85,B 0,C 180,E1 -17506.933,E2 -17506.933} C_VEL
LIN {X 0,Y 282.545,Z 312.301,A -85,B 0,C 180,E1 -17507.467,E2 -17507.467} C_VEL
LIN {X 0,Y 288.937,Z 321.928,A -85,B 0,C 180,E1 -17508.941,E2 -17508.941} C_VEL
LIN {X 0,Y 293.214,Z 328.943,A -85,B 0,C 180,E1 -17509.892,E2 -17509.892} C_VEL
LIN {X 0,Y 300.721,Z 343.195,A -85,B 0,C 180,E1 -17511.524,E2 -17511.524} C_VEL
LIN {X 0,Y 308.038,Z 358.92,A -85,B 0,C 180,E1 -17513.059,E2 -17513.059} C_VEL
LIN {X 0,Y 308.489,Z 359.917,A -85,B 0,C 180,E1 -17513.151,E2 -17513.151} C_VEL
LIN {X 0,Y 304.257,Z 463.309,A -85,B 0,C 180,E1 -17515.535,E2 -17515.535} C_VEL
LIN {X 0,Y 303.03,Z 478.679,A -85,B 0,C 180,E1 -17516.079,E2 -17516.079} C_VEL
LIN {X 0,Y 301.443,Z 493.287,A -85,B 0,C 180,E1 -17516.858,E2 -17516.858} C_VEL
LIN {X 0,Y 299.54,Z 506.779,A -85,B 0,C 180,E1 -17517.819,E2 -17517.819} C_VEL
LIN {X 0,Y 297.265,Z 520.353,A -85,B 0,C 180,E1 -17519.056,E2 -17519.056} C_VEL
LIN {X 0,Y 294.543,Z 533.407,A -85,B 0,C 180,E1 -17520.52,E2 -17520.52} C_VEL
LIN {X 0,Y 291.821,Z 545.421,A -85,B 0,C 180,E1 -17522.186,E2 -17522.186} C_VEL
LIN {X 0,Y 288.96,Z 556.52,A -85,B 0,C 180,E1 -17524.038,E2 -17524.038} C_VEL
LIN {X 0,Y 286.362,Z 566.695,A -85,B 0,C 180,E1 -17526.113,E2 -17526.113} C_VEL
LIN {X 0,Y 283.574,Z 576.651,A -85,B 0,C 180,E1 -17528.559,E2 -17528.559} C_VEL
LIN {X 0,Y 281.2,Z 584.905,A -85,B 0,C 180,E1 -17531.041,E2 -17531.041} C_VEL
LIN {X 0,Y 279.117,Z 592.651,A -85,B 0,C 180,E1 -17533.921,E2 -17533.921} C_VEL
LIN {X 0,Y 277.491,Z 598.814,A -85,B 0,C 180,E1 -17536.824,E2 -17536.824} C_VEL
LIN {X 0,Y 276.469,Z 603.566,A -85,B 0,C 180,E1 -17539.75,E2 -17539.75} C_VEL
LIN {X 0,Y 275.822,Z 607.044,A -85,B 0,C 180,E1 -17542.681,E2 -17542.681} C_VEL
LIN {X 0,Y 275.472,Z 609.341,A -85,B 0,C 180,E1 -17545.611,E2 -17545.611} C_VEL
LIN {X 0,Y 275.297,Z 610.513,A -85,B 0,C 180,E1 -17548.537,E2 -17548.537} C_VEL
LIN {X 0,Y 275.297,Z 610.526,A -85,B 0,C 180,E1 -17551.463,E2 -17551.463} C_VEL
LIN {X 0,Y 275.464,Z 609.409,A -85,B 0,C 180,E1 -17554.39,E2 -17554.39} C_VEL
LIN {X 0,Y 275.777,Z 607.164,A -85,B 0,C 180,E1 -17557.32,E2 -17557.32} C_VEL
LIN {X 0,Y 276.447,Z 603.733,A -85,B 0,C 180,E1 -17560.251,E2 -17560.251} C_VEL
LIN {X 0,Y 277.461,Z 599.034,A -85,B 0,C 180,E1 -17563.177,E2 -17563.177} C_VEL
LIN {X 0,Y 279.094,Z 592.938,A -85,B 0,C 180,E1 -17566.081,E2 -17566.081} C_VEL
LIN {X 0,Y 281.132,Z 585.261,A -85,B 0,C 180,E1 -17568.964,E2 -17568.964} C_VEL
LIN {X 0,Y 283.475,Z 577.069,A -85,B 0,C 180,E1 -17571.449,E2 -17571.449} C_VEL
LIN {X 0,Y 286.284,Z 567.195,A -85,B 0,C 180,E1 -17573.894,E2 -17573.894} C_VEL
LIN {X 0,Y 288.885,Z 557.074,A -85,B 0,C 180,E1 -17575.97,E2 -17575.97} C_VEL
LIN {X 0,Y 291.707,Z 546.075,A -85,B 0,C 180,E1 -17577.826,E2 -17577.826} C_VEL
LIN {X 0,Y 294.407,Z 534.199,A -85,B 0,C 180,E1 -17579.495,E2 -17579.495} C_VEL
LIN {X 0,Y 297.115,Z 521.335,A -85,B 0,C 180,E1 -17580.962,E2 -17580.962} C_VEL
LIN {X 0,Y 299.617,Z 506.98,A -85,B 0,C 180,E1 -17582.275,E2 -17582.275} C_VEL
LIN {X 0,Y 301.604,Z 492.535,A -85,B 0,C 180,E1 -17583.301,E2 -17583.301} C_VEL
LIN {X 0,Y 303.252,Z 477.252,A -85,B 0,C 180,E1 -17584.093,E2 -17584.093} C_VEL
LIN {X 0,Y 304.38,Z 462.484,A -85,B 0,C 180,E1 -17584.6,E2 -17584.6} C_VEL
LIN {X 0,Y 308.584,Z 360.88,A -85,B 0,C 180,E1 -17586.933,E2 -17586.933} C_VEL
LIN {X 0,Y 308.32,Z 359.456,A -85,B 0,C 180,E1 -17587.011,E2 -17587.011} C_VEL
LIN {X 0,Y 301.165,Z 344.064,A -85,B 0,C 180,E1 -17588.51,E2 -17588.51} C_VEL
LIN {X 0,Y 294.15,Z 330.509,A -85,B 0,C 180,E1 -17590.036,E2 -17590.036} C_VEL
LIN {X 0,Y 287.969,Z 320.326,A -85,B 0,C 180,E1 -17591.416,E2 -17591.416} C_VEL
LIN {X 0,Y 282.412,Z 312.174,A -85,B 0,C 180,E1 -17592.701,E2 -17592.701} C_VEL
LIN {X 0,Y 280.219,Z 308.692,A -85,B 0,C 180,E1 -17593.239,E2 -17593.239} C_VEL
LIN {X 0,Y 277.923,Z 305.9,A -85,B 0,C 180,E1 -17593.786,E2 -17593.786} C_VEL
LIN {X 0,Y 277.206,Z 303.582,A -85,B 0,C 180,E1 -17594.046,E2 -17594.046} C_VEL
LIN {X 0,Y 277.196,Z 303.579,A -85,B 0,C 180,E1 -17594.955,E2 -17594.955} C_VEL
LIN {X 0,Y 276.551,Z 303.664,A -85,B 0,C 180,E1 -17596.168,E2 -17596.168} C_VEL
LIN {X 0,Y 273.766,Z 304.021,A -85,B 0,C 180,E1 -17598.147,E2 -17598.147} C_VEL
LIN {X 0,Y 271.373,Z 304.319,A -85,B 0,C 180,E1 -17599.754,E2 -17599.754} C_VEL
LIN {X 0,Y 270.307,Z 304.439,A -85,B 0,C 180,E1 -17600.998,E2 -17600.998} C_VEL
LIN {X 0,Y 270.2,Z 304.445,A -85,B 0,C 180,E1 -17601.419,E2 -17601.419} C_VEL
LIN {X 0,Y 270.193,Z 304.444,A -85,B 0,C 180,E1 -17605.093,E2 -17605.093} C_VEL
LIN {X 0,Y 270.179,Z 304.423,A -85,B 0,C 180,E1 -17609.136,E2 -17609.136} C_VEL
LIN {X 0,Y 270.254,Z 304.445,A -85,B 0,C 180,E1 -17612.147,E2 -17612.147} C_VEL
LIN {X 0,Y 270.227,Z 304.446,A -85,B 0,C 180,E1 -17615.539,E2 -17615.539} C_VEL
LIN {X 0,Y 270.251,Z 304.447,A -85,B 0,C 180,E1 -17620.24,E2 -17620.24} C_VEL
LIN {X 0,Y 270.361,Z 304.432,A -85,B 0,C 180,E1 -17624.933,E2 -17624.933} C_VEL
LIN {X 0,Y 270.402,Z 304.425,A -85,B 0,C 180,E1 -17629.517,E2 -17629.517} C_VEL
LIN {X 0,Y 270.566,Z 304.404,A -85,B 0,C 180,E1 -17632.537,E2 -17632.537} C_VEL
LIN {X 0,Y 270.771,Z 304.38,A -85,B 0,C 180,E1 -17638.513,E2 -17638.513} C_VEL
LIN {X 0,Y 270.767,Z 304.379,A -85,B 0,C 180,E1 -17641.487,E2 -17641.487} C_VEL
LIN {X 0,Y 270.561,Z 304.408,A -85,B 0,C 180,E1 -17647.462,E2 -17647.462} C_VEL
LIN {X 0,Y 270.402,Z 304.425,A -85,B 0,C 180,E1 -17650.482,E2 -17650.482} C_VEL
LIN {X 0,Y 270.36,Z 304.434,A -85,B 0,C 180,E1 -17655.067,E2 -17655.067} C_VEL
LIN {X 0,Y 270.215,Z 304.454,A -85,B 0,C 180,E1 -17659.762,E2 -17659.762} C_VEL
LIN {X 0,Y 270.177,Z 304.457,A -85,B 0,C 180,E1 -17664.437,E2 -17664.437} C_VEL
LIN {X 0,Y 270.19,Z 304.457,A -85,B 0,C 180,E1 -17667.918,E2 -17667.918} C_VEL
LIN {X 0,Y 270.167,Z 304.458,A -85,B 0,C 180,E1 -17671.35,E2 -17671.35} C_VEL
LIN {X 0,Y 270.191,Z 304.454,A -85,B 0,C 180,E1 -17674.907,E2 -17674.907} C_VEL
LIN {X 0,Y 270.162,Z 304.447,A -85,B 0,C 180,E1 -17678.703,E2 -17678.703} C_VEL
LIN {X 0,Y 270.125,Z 304.464,A -85,B 0,C 180,E1 -17681.622,E2 -17681.622} C_VEL
LIN {X 0,Y 272.869,Z 312.921,A -85,B 0,C 180,E1 -17685.079,E2 -17685.079} C_VEL
LIN {X 0,Y 275.681,Z 317.543,A -85,B 0,C 180,E1 -17685.82,E2 -17685.82} C_VEL
LIN {X 0,Y 281.95,Z 328.098,A -85,B 0,C 180,E1 -17687.395,E2 -17687.395} C_VEL
LIN {X 0,Y 290.146,Z 343.329,A -85,B 0,C 180,E1 -17689.345,E2 -17689.345} C_VEL
LIN {X 0,Y 297.281,Z 358.284,A -85,B 0,C 180,E1 -17690.964,E2 -17690.964} C_VEL
LIN {X 0,Y 301.888,Z 369.211,A -85,B 0,C 180,E1 -17691.988,E2 -17691.988} C_VEL
LIN {X 0,Y 302.485,Z 374.307,A -85,B 0,C 180,E1 -17692.226,E2 -17692.226} C_VEL
LIN {X 0,Y 298.054,Z 476.768,A -85,B 0,C 180,E1 -17694.609,E2 -17694.609} C_VEL
LIN {X 0,Y 296.774,Z 492.415,A -85,B 0,C 180,E1 -17695.159,E2 -17695.159} C_VEL
LIN {X 0,Y 294.842,Z 507.448,A -85,B 0,C 180,E1 -17695.934,E2 -17695.934} C_VEL
LIN {X 0,Y 292.717,Z 521.034,A -85,B 0,C 180,E1 -17696.894,E2 -17696.894} C_VEL
LIN {X 0,Y 290.196,Z 534.4,A -85,B 0,C 180,E1 -17698.098,E2 -17698.098} C_VEL
LIN {X 0,Y 287.117,Z 548.321,A -85,B 0,C 180,E1 -17699.679,E2 -17699.679} C_VEL
LIN {X 0,Y 283.834,Z 561.412,A -85,B 0,C 180,E1 -17701.534,E2 -17701.534} C_VEL
LIN {X 0,Y 280.649,Z 573.266,A -85,B 0,C 180,E1 -17703.61,E2 -17703.61} C_VEL
LIN {X 0,Y 277.889,Z 583.158,A -85,B 0,C 180,E1 -17705.711,E2 -17705.711} C_VEL
LIN {X 0,Y 275.561,Z 591.761,A -85,B 0,C 180,E1 -17707.903,E2 -17707.903} C_VEL
LIN {X 0,Y 273.144,Z 600.092,A -85,B 0,C 180,E1 -17710.459,E2 -17710.459} C_VEL
LIN {X 0,Y 271.095,Z 607.928,A -85,B 0,C 180,E1 -17713.431,E2 -17713.431} C_VEL
LIN {X 0,Y 269.677,Z 614.169,A -85,B 0,C 180,E1 -17716.435,E2 -17716.435} C_VEL
LIN {X 0,Y 268.723,Z 619,A -85,B 0,C 180,E1 -17719.451,E2 -17719.451} C_VEL
LIN {X 0,Y 268.28,Z 622.545,A -85,B 0,C 180,E1 -17722.474,E2 -17722.474} C_VEL
LIN {X 0,Y 268.107,Z 624.879,A -85,B 0,C 180,E1 -17725.49,E2 -17725.49} C_VEL
LIN {X 0,Y 268.182,Z 626.055,A -85,B 0,C 180,E1 -17728.498,E2 -17728.498} C_VEL
LIN {X 0,Y 268.182,Z 626.051,A -85,B 0,C 180,E1 -17731.502,E2 -17731.502} C_VEL
LIN {X 0,Y 268.107,Z 624.86,A -85,B 0,C 180,E1 -17734.51,E2 -17734.51} C_VEL
LIN {X 0,Y 268.237,Z 622.512,A -85,B 0,C 180,E1 -17737.527,E2 -17737.527} C_VEL
LIN {X 0,Y 268.709,Z 618.961,A -85,B 0,C 180,E1 -17740.549,E2 -17740.549} C_VEL
LIN {X 0,Y 269.671,Z 614.119,A -85,B 0,C 180,E1 -17743.565,E2 -17743.565} C_VEL
LIN {X 0,Y 271.002,Z 607.852,A -85,B 0,C 180,E1 -17746.574,E2 -17746.574} C_VEL
LIN {X 0,Y 273.17,Z 600,A -85,B 0,C 180,E1 -17749.539,E2 -17749.539} C_VEL
LIN {X 0,Y 275.575,Z 591.655,A -85,B 0,C 180,E1 -17752.096,E2 -17752.096} C_VEL
LIN {X 0,Y 278.377,Z 581.464,A -85,B 0,C 180,E1 -17754.651,E2 -17754.651} C_VEL
LIN {X 0,Y 281.134,Z 571.331,A -85,B 0,C 180,E1 -17756.741,E2 -17756.741} C_VEL
LIN {X 0,Y 284.431,Z 559.097,A -85,B 0,C 180,E1 -17758.804,E2 -17758.804} C_VEL
LIN {X 0,Y 287.434,Z 546.82,A -85,B 0,C 180,E1 -17760.487,E2 -17760.487} C_VEL
LIN {X 0,Y 290.363,Z 533.083,A -85,B 0,C 180,E1 -17762.016,E2 -17762.016} C_VEL
LIN {X 0,Y 293.049,Z 518.706,A -85,B 0,C 180,E1 -17763.269,E2 -17763.269} C_VEL
LIN {X 0,Y 295.236,Z 504.422,A -85,B 0,C 180,E1 -17764.22,E2 -17764.22} C_VEL
LIN {X 0,Y 296.969,Z 489.979,A -85,B 0,C 180,E1 -17764.918,E2 -17764.918} C_VEL
LIN {X 0,Y 298.009,Z 475.747,A -85,B 0,C 180,E1 -17765.397,E2 -17765.397} C_VEL
LIN {X 0,Y 302.411,Z 374.049,A -85,B 0,C 180,E1 -17767.756,E2 -17767.756} C_VEL
LIN {X 0,Y 301.513,Z 368.334,A -85,B 0,C 180,E1 -17768.056,E2 -17768.056} C_VEL
LIN {X 0,Y 294.34,Z 351.917,A -85,B 0,C 180,E1 -17769.655,E2 -17769.655} C_VEL
LIN {X 0,Y 287.61,Z 338.515,A -85,B 0,C 180,E1 -17771.199,E2 -17771.199} C_VEL
LIN {X 0,Y 281.161,Z 326.827,A -85,B 0,C 180,E1 -17772.746,E2 -17772.746} C_VEL
LIN {X 0,Y 277.62,Z 320.891,A -85,B 0,C 180,E1 -17773.627,E2 -17773.627} C_VEL
LIN {X 0,Y 274.684,Z 316.12,A -85,B 0,C 180,E1 -17774.379,E2 -17774.379} C_VEL
LIN {X 0,Y 272.714,Z 312.608,A -85,B 0,C 180,E1 -17774.951,E2 -17774.951} C_VEL
LIN {X 0,Y 270.126,Z 304.465,A -85,B 0,C 180,E1 -17778.378,E2 -17778.378} C_VEL
LIN {X 0,Y 270.147,Z 304.456,A -85,B 0,C 180,E1 -17781.364,E2 -17781.364} C_VEL
LIN {X 0,Y 270.191,Z 304.449,A -85,B 0,C 180,E1 -17785.093,E2 -17785.093} C_VEL
LIN {X 0,Y 270.178,Z 304.453,A -85,B 0,C 180,E1 -17789.136,E2 -17789.136} C_VEL
LIN {X 0,Y 270.184,Z 304.451,A -85,B 0,C 180,E1 -17792.175,E2 -17792.175} C_VEL
LIN {X 0,Y 270.175,Z 304.451,A -85,B 0,C 180,E1 -17795.564,E2 -17795.564} C_VEL
LIN {X 0,Y 270.215,Z 304.421,A -85,B 0,C 180,E1 -17800.238,E2 -17800.238} C_VEL
LIN {X 0,Y 270.36,Z 304.433,A -85,B 0,C 180,E1 -17804.933,E2 -17804.933} C_VEL
LIN {X 0,Y 270.378,Z 304.395,A -85,B 0,C 180,E1 -17809.517,E2 -17809.517} C_VEL
LIN {X 0,Y 270.546,Z 304.41,A -85,B 0,C 180,E1 -17812.537,E2 -17812.537} C_VEL
LIN {X 0,Y 270.767,Z 304.372,A -85,B 0,C 180,E1 -17818.513,E2 -17818.513} C_VEL
LIN {X 0,Y 270.762,Z 304.379,A -85,B 0,C 180,E1 -17821.488,E2 -17821.488} C_VEL
LIN {X 0,Y 270.562,Z 304.4,A -85,B 0,C 180,E1 -17827.463,E2 -17827.463} C_VEL
LIN {X 0,Y 270.38,Z 304.423,A -85,B 0,C 180,E1 -17830.484,E2 -17830.484} C_VEL
LIN {X 0,Y 270.36,Z 304.425,A -85,B 0,C 180,E1 -17835.067,E2 -17835.067} C_VEL
LIN {X 0,Y 270.217,Z 304.419,A -85,B 0,C 180,E1 -17839.762,E2 -17839.762} C_VEL
LIN {X 0,Y 270.227,Z 304.45,A -85,B 0,C 180,E1 -17844.59,E2 -17844.59} C_VEL
LIN {X 0,Y 270.238,Z 304.42,A -85,B 0,C 180,E1 -17847.913,E2 -17847.913} C_VEL
LIN {X 0,Y 270.179,Z 304.451,A -85,B 0,C 180,E1 -17851.349,E2 -17851.349} C_VEL
LIN {X 0,Y 270.196,Z 304.448,A -85,B 0,C 180,E1 -17854.907,E2 -17854.907} C_VEL
LIN {X 0,Y 270.194,Z 304.452,A -85,B 0,C 180,E1 -17858.711,E2 -17858.711} C_VEL
LIN {X 0,Y 270.161,Z 304.456,A -85,B 0,C 180,E1 -17863.25,E2 -17863.25} C_VEL
LIN {X 0,Y 270.16,Z 304.485,A -85,B 0,C 180,E1 -17864.699,E2 -17864.699} C_VEL
LIN {X 0,Y 271.058,Z 307.128,A -85,B 0,C 180,E1 -17864.989,E2 -17864.989} C_VEL
LIN {X 0,Y 273.49,Z 310.105,A -85,B 0,C 180,E1 -17865.608,E2 -17865.608} C_VEL
LIN {X 0,Y 275.723,Z 313.39,A -85,B 0,C 180,E1 -17866.181,E2 -17866.181} C_VEL
LIN {X 0,Y 282.79,Z 323.834,A -85,B 0,C 180,E1 -17867.903,E2 -17867.903} C_VEL
LIN {X 0,Y 288.361,Z 332.756,A -85,B 0,C 180,E1 -17869.192,E2 -17869.192} C_VEL
LIN {X 0,Y 296.859,Z 349.168,A -85,B 0,C 180,E1 -17871.107,E2 -17871.107} C_VEL
LIN {X 0,Y 302.749,Z 362.094,A -85,B 0,C 180,E1 -17872.389,E2 -17872.389} C_VEL
LIN {X 0,Y 298.887,Z 453.736,A -85,B 0,C 180,E1 -17874.516,E2 -17874.516} C_VEL
LIN {X 0,Y 297.908,Z 471.005,A -85,B 0,C 180,E1 -17875.002,E2 -17875.002} C_VEL
LIN {X 0,Y 296.418,Z 486.19,A -85,B 0,C 180,E1 -17875.679,E2 -17875.679} C_VEL
LIN {X 0,Y 294.504,Z 500.886,A -85,B 0,C 180,E1 -17876.609,E2 -17876.609} C_VEL
LIN {X 0,Y 292.356,Z 514.569,A -85,B 0,C 180,E1 -17877.756,E2 -17877.756} C_VEL
LIN {X 0,Y 289.567,Z 528.12,A -85,B 0,C 180,E1 -17879.156,E2 -17879.156} C_VEL
LIN {X 0,Y 286.669,Z 541.055,A -85,B 0,C 180,E1 -17880.84,E2 -17880.84} C_VEL
LIN {X 0,Y 283.626,Z 552.866,A -85,B 0,C 180,E1 -17882.716,E2 -17882.716} C_VEL
LIN {X 0,Y 281.231,Z 562.068,A -85,B 0,C 180,E1 -17884.472,E2 -17884.472} C_VEL
LIN {X 0,Y 278.114,Z 572.826,A -85,B 0,C 180,E1 -17886.941,E2 -17886.941} C_VEL
LIN {X 0,Y 275.51,Z 581.779,A -85,B 0,C 180,E1 -17889.467,E2 -17889.467} C_VEL
LIN {X 0,Y 273.164,Z 589.579,A -85,B 0,C 180,E1 -17892.165,E2 -17892.165} C_VEL
LIN {X 0,Y 271.41,Z 596.122,A -85,B 0,C 180,E1 -17894.993,E2 -17894.993} C_VEL
LIN {X 0,Y 269.96,Z 601.561,A -85,B 0,C 180,E1 -17897.98,E2 -17897.98} C_VEL
LIN {X 0,Y 269.089,Z 605.661,A -85,B 0,C 180,E1 -17900.984,E2 -17900.984} C_VEL
LIN {X 0,Y 268.494,Z 608.612,A -85,B 0,C 180,E1 -17904.087,E2 -17904.087} C_VEL
LIN {X 0,Y 268.308,Z 610.268,A -85,B 0,C 180,E1 -17906.997,E2 -17906.997} C_VEL
LIN {X 0,Y 268.207,Z 610.872,A -85,B 0,C 180,E1 -17910,E2 -17910} C_VEL
LIN {X 0,Y 268.305,Z 610.308,A -85,B 0,C 180,E1 -17913.003,E2 -17913.003} C_VEL
LIN {X 0,Y 268.505,Z 608.633,A -85,B 0,C 180,E1 -17916.01,E2 -17916.01} C_VEL
LIN {X 0,Y 269.022,Z 605.804,A -85,B 0,C 180,E1 -17919.018,E2 -17919.018} C_VEL
LIN {X 0,Y 269.932,Z 601.751,A -85,B 0,C 180,E1 -17922.022,E2 -17922.022} C_VEL
LIN {X 0,Y 271.379,Z 596.371,A -85,B 0,C 180,E1 -17925.009,E2 -17925.009} C_VEL
LIN {X 0,Y 273.247,Z 589.515,A -85,B 0,C 180,E1 -17927.977,E2 -17927.977} C_VEL
LIN {X 0,Y 275.756,Z 580.949,A -85,B 0,C 180,E1 -17930.904,E2 -17930.904} C_VEL
LIN {X 0,Y 278.41,Z 571.837,A -85,B 0,C 180,E1 -17933.426,E2 -17933.426} C_VEL
LIN {X 0,Y 280.997,Z 562.88,A -85,B 0,C 180,E1 -17935.477,E2 -17935.477} C_VEL
LIN {X 0,Y 284.025,Z 551.519,A -85,B 0,C 180,E1 -17937.642,E2 -17937.642} C_VEL
LIN {X 0,Y 287.142,Z 539.427,A -85,B 0,C 180,E1 -17939.509,E2 -17939.509} C_VEL
LIN {X 0,Y 289.824,Z 527.566,A -85,B 0,C 180,E1 -17941.016,E2 -17941.016} C_VEL
LIN {X 0,Y 292.406,Z 514.651,A -85,B 0,C 180,E1 -17942.354,E2 -17942.354} C_VEL
LIN {X 0,Y 294.573,Z 501.128,A -85,B 0,C 180,E1 -17943.484,E2 -17943.484} C_VEL
LIN {X 0,Y 296.455,Z 486.501,A -85,B 0,C 180,E1 -17944.419,E2 -17944.419} C_VEL
LIN {X 0,Y 297.992,Z 471.48,A -85,B 0,C 180,E1 -17945.09,E2 -17945.09} C_VEL
LIN {X 0,Y 298.993,Z 454.494,A -85,B 0,C 180,E1 -17945.573,E2 -17945.573} C_VEL
LIN {X 0,Y 302.849,Z 362.172,A -85,B 0,C 180,E1 -17947.72,E2 -17947.72} C_VEL
LIN {X 0,Y 295.366,Z 346.098,A -85,B 0,C 180,E1 -17949.354,E2 -17949.354} C_VEL
LIN {X 0,Y 288.98,Z 333.829,A -85,B 0,C 180,E1 -17950.801,E2 -17950.801} C_VEL
LIN {X 0,Y 283.178,Z 324.395,A -85,B 0,C 180,E1 -17952.145,E2 -17952.145} C_VEL
LIN {X 0,Y 277.606,Z 316.215,A -85,B 0,C 180,E1 -17953.487,E2 -17953.487} C_VEL
LIN {X 0,Y 275.53,Z 313.191,A -85,B 0,C 180,E1 -17954.008,E2 -17954.008} C_VEL
LIN {X 0,Y 273.395,Z 309.927,A -85,B 0,C 180,E1 -17954.563,E2 -17954.563} C_VEL
LIN {X 0,Y 270.868,Z 306.795,A -85,B 0,C 180,E1 -17955.211,E2 -17955.211} C_VEL
LIN {X 0,Y 270.167,Z 304.456,A -85,B 0,C 180,E1 -17955.477,E2 -17955.477} C_VEL
LIN {X 0,Y 270.169,Z 304.443,A -85,B 0,C 180,E1 -17959.433,E2 -17959.433} C_VEL
LIN {X 0,Y 270.2,Z 304.445,A -85,B 0,C 180,E1 -17961.419,E2 -17961.419} C_VEL
LIN {X 0,Y 269.479,Z 304.522,A -85,B 0,C 180,E1 -17962.663,E2 -17962.663} C_VEL
LIN {X 0,Y 266.618,Z 304.882,A -85,B 0,C 180,E1 -17964.691,E2 -17964.691} C_VEL
LIN {X 0,Y 264.224,Z 305.198,A -85,B 0,C 180,E1 -17966.339,E2 -17966.339} C_VEL
LIN {X 0,Y 263.199,Z 305.307,A -85,B 0,C 180,E1 -17967.616,E2 -17967.616} C_VEL
LIN {X 0,Y 263.114,Z 305.311,A -85,B 0,C 180,E1 -17968.049,E2 -17968.049} C_VEL
LIN {X 0,Y 263.172,Z 305.322,A -85,B 0,C 180,E1 -17971.792,E2 -17971.792} C_VEL
LIN {X 0,Y 263.191,Z 305.32,A -85,B 0,C 180,E1 -17975.213,E2 -17975.213} C_VEL
LIN {X 0,Y 263.231,Z 305.321,A -85,B 0,C 180,E1 -17979.691,E2 -17979.691} C_VEL
LIN {X 0,Y 263.303,Z 305.313,A -85,B 0,C 180,E1 -17984.519,E2 -17984.519} C_VEL
LIN {X 0,Y 263.342,Z 305.306,A -85,B 0,C 180,E1 -17989.233,E2 -17989.233} C_VEL
LIN {X 0,Y 263.528,Z 305.279,A -85,B 0,C 180,E1 -17992.337,E2 -17992.337} C_VEL
LIN {X 0,Y 263.734,Z 305.257,A -85,B 0,C 180,E1 -17998.473,E2 -17998.473} C_VEL
LIN {X 0,Y 263.731,Z 305.256,A -85,B 0,C 180,E1 -18001.527,E2 -18001.527} C_VEL
LIN {X 0,Y 263.524,Z 305.284,A -85,B 0,C 180,E1 -18007.663,E2 -18007.663} C_VEL
LIN {X 0,Y 263.341,Z 305.307,A -85,B 0,C 180,E1 -18010.767,E2 -18010.767} C_VEL
LIN {X 0,Y 263.303,Z 305.315,A -85,B 0,C 180,E1 -18015.481,E2 -18015.481} C_VEL
LIN {X 0,Y 263.201,Z 305.327,A -85,B 0,C 180,E1 -18020.311,E2 -18020.311} C_VEL
LIN {X 0,Y 263.12,Z 305.329,A -85,B 0,C 180,E1 -18025.3,E2 -18025.3} C_VEL
LIN {X 0,Y 263.123,Z 305.334,A -85,B 0,C 180,E1 -18028.736,E2 -18028.736} C_VEL
LIN {X 0,Y 263.122,Z 305.328,A -85,B 0,C 180,E1 -18032.29,E2 -18032.29} C_VEL
LIN {X 0,Y 263.167,Z 305.322,A -85,B 0,C 180,E1 -18036.761,E2 -18036.761} C_VEL
LIN {X 0,Y 263.109,Z 305.489,A -85,B 0,C 180,E1 -18040.372,E2 -18040.372} C_VEL
LIN {X 0,Y 265.405,Z 312.54,A -85,B 0,C 180,E1 -18043.445,E2 -18043.445} C_VEL
LIN {X 0,Y 268.521,Z 317.451,A -85,B 0,C 180,E1 -18044.322,E2 -18044.322} C_VEL
LIN {X 0,Y 276.053,Z 330.037,A -85,B 0,C 180,E1 -18046.335,E2 -18046.335} C_VEL
LIN {X 0,Y 283.063,Z 342.822,A -85,B 0,C 180,E1 -18048.093,E2 -18048.093} C_VEL
LIN {X 0,Y 289.902,Z 356.677,A -85,B 0,C 180,E1 -18049.729,E2 -18049.729} C_VEL
LIN {X 0,Y 296.529,Z 372.108,A -85,B 0,C 180,E1 -18051.268,E2 -18051.268} C_VEL
LIN {X 0,Y 296.824,Z 375.922,A -85,B 0,C 180,E1 -18051.429,E2 -18051.429} C_VEL
LIN {X 0,Y 292.217,Z 478.089,A -85,B 0,C 180,E1 -18053.845,E2 -18053.845} C_VEL
LIN {X 0,Y 290.873,Z 493.139,A -85,B 0,C 180,E1 -18054.399,E2 -18054.399} C_VEL
LIN {X 0,Y 288.815,Z 508.556,A -85,B 0,C 180,E1 -18055.228,E2 -18055.228} C_VEL
LIN {X 0,Y 286.417,Z 522.825,A -85,B 0,C 180,E1 -18056.279,E2 -18056.279} C_VEL
LIN {X 0,Y 283.977,Z 535.129,A -85,B 0,C 180,E1 -18057.437,E2 -18057.437} C_VEL
LIN {X 0,Y 280.997,Z 548.121,A -85,B 0,C 180,E1 -18058.947,E2 -18058.947} C_VEL
LIN {X 0,Y 277.598,Z 561.211,A -85,B 0,C 180,E1 -18060.834,E2 -18060.834} C_VEL
LIN {X 0,Y 274.243,Z 573.063,A -85,B 0,C 180,E1 -18062.944,E2 -18062.944} C_VEL
LIN {X 0,Y 271.169,Z 583.624,A -85,B 0,C 180,E1 -18065.252,E2 -18065.252} C_VEL
LIN {X 0,Y 268.531,Z 592.816,A -85,B 0,C 180,E1 -18067.698,E2 -18067.698} C_VEL
LIN {X 0,Y 266.067,Z 600.971,A -85,B 0,C 180,E1 -18070.32,E2 -18070.32} C_VEL
LIN {X 0,Y 263.984,Z 608.69,A -85,B 0,C 180,E1 -18073.419,E2 -18073.419} C_VEL
LIN {X 0,Y 262.41,Z 615.292,A -85,B 0,C 180,E1 -18076.842,E2 -18076.842} C_VEL
LIN {X 0,Y 261.688,Z 618.796,A -85,B 0,C 180,E1 -18079.165,E2 -18079.165} C_VEL
LIN {X 0,Y 261.201,Z 622.341,A -85,B 0,C 180,E1 -18082.269,E2 -18082.269} C_VEL
LIN {X 0,Y 261.017,Z 624.676,A -85,B 0,C 180,E1 -18085.367,E2 -18085.367} C_VEL
LIN {X 0,Y 261.109,Z 625.853,A -85,B 0,C 180,E1 -18088.458,E2 -18088.458} C_VEL
LIN {X 0,Y 261.109,Z 625.849,A -85,B 0,C 180,E1 -18091.542,E2 -18091.542} C_VEL
LIN {X 0,Y 261.084,Z 624.388,A -85,B 0,C 180,E1 -18095.137,E2 -18095.137} C_VEL
LIN {X 0,Y 261.151,Z 622.307,A -85,B 0,C 180,E1 -18097.733,E2 -18097.733} C_VEL
LIN {X 0,Y 261.676,Z 618.755,A -85,B 0,C 180,E1 -18100.836,E2 -18100.836} C_VEL
LIN {X 0,Y 262.691,Z 613.912,A -85,B 0,C 180,E1 -18103.932,E2 -18103.932} C_VEL
LIN {X 0,Y 264.155,Z 607.646,A -85,B 0,C 180,E1 -18107.017,E2 -18107.017} C_VEL
LIN {X 0,Y 266.4,Z 599.792,A -85,B 0,C 180,E1 -18110.057,E2 -18110.057} C_VEL
LIN {X 0,Y 268.953,Z 591.448,A -85,B 0,C 180,E1 -18112.67,E2 -18112.67} C_VEL
LIN {X 0,Y 271.717,Z 581.873,A -85,B 0,C 180,E1 -18115.139,E2 -18115.139} C_VEL
LIN {X 0,Y 274.786,Z 571.125,A -85,B 0,C 180,E1 -18117.41,E2 -18117.41} C_VEL
LIN {X 0,Y 278.19,Z 558.889,A -85,B 0,C 180,E1 -18119.513,E2 -18119.513} C_VEL
LIN {X 0,Y 281.323,Z 546.612,A -85,B 0,C 180,E1 -18121.222,E2 -18121.222} C_VEL
LIN {X 0,Y 284.367,Z 532.742,A -85,B 0,C 180,E1 -18122.792,E2 -18122.792} C_VEL
LIN {X 0,Y 287.12,Z 518.495,A -85,B 0,C 180,E1 -18124.049,E2 -18124.049} C_VEL
LIN {X 0,Y 289.399,Z 504.212,A -85,B 0,C 180,E1 -18125.009,E2 -18125.009} C_VEL
LIN {X 0,Y 291.179,Z 489.765,A -85,B 0,C 180,E1 -18125.717,E2 -18125.717} C_VEL
LIN {X 0,Y 292.261,Z 475.526,A -85,B 0,C 180,E1 -18126.202,E2 -18126.202} C_VEL
LIN {X 0,Y 296.74,Z 375.731,A -85,B 0,C 180,E1 -18128.551,E2 -18128.551} C_VEL
LIN {X 0,Y 296.408,Z 371.91,A -85,B 0,C 180,E1 -18128.718,E2 -18128.718} C_VEL
LIN {X 0,Y 289.425,Z 355.69,A -85,B 0,C 180,E1 -18130.34,E2 -18130.34} C_VEL
LIN {X 0,Y 282.001,Z 340.766,A -85,B 0,C 180,E1 -18132.121,E2 -18132.121} C_VEL
LIN {X 0,Y 273.959,Z 326.496,A -85,B 0,C 180,E1 -18134.155,E2 -18134.155} C_VEL
LIN {X 0,Y 268.066,Z 316.909,A -85,B 0,C 180,E1 -18135.739,E2 -18135.739} C_VEL
LIN {X 0,Y 265.346,Z 312.358,A -85,B 0,C 180,E1 -18136.543,E2 -18136.543} C_VEL
LIN {X 0,Y 263.091,Z 305.335,A -85,B 0,C 180,E1 -18139.687,E2 -18139.687} C_VEL
LIN {X 0,Y 263.147,Z 305.326,A -85,B 0,C 180,E1 -18144.016,E2 -18144.016} C_VEL
LIN {X 0,Y 263.122,Z 305.329,A -85,B 0,C 180,E1 -18147.71,E2 -18147.71} C_VEL
LIN {X 0,Y 263.134,Z 305.332,A -85,B 0,C 180,E1 -18151.808,E2 -18151.808} C_VEL
LIN {X 0,Y 263.108,Z 305.331,A -85,B 0,C 180,E1 -18156.38,E2 -18156.38} C_VEL
LIN {X 0,Y 263.201,Z 305.3,A -85,B 0,C 180,E1 -18159.689,E2 -18159.689} C_VEL
LIN {X 0,Y 263.303,Z 305.312,A -85,B 0,C 180,E1 -18164.519,E2 -18164.519} C_VEL
LIN {X 0,Y 263.324,Z 305.271,A -85,B 0,C 180,E1 -18169.233,E2 -18169.233} C_VEL
LIN {X 0,Y 263.508,Z 305.286,A -85,B 0,C 180,E1 -18172.337,E2 -18172.337} C_VEL
LIN {X 0,Y 263.73,Z 305.248,A -85,B 0,C 180,E1 -18178.473,E2 -18178.473} C_VEL
LIN {X 0,Y 263.726,Z 305.255,A -85,B 0,C 180,E1 -18181.527,E2 -18181.527} C_VEL
LIN {X 0,Y 263.524,Z 305.278,A -85,B 0,C 180,E1 -18187.663,E2 -18187.663} C_VEL
LIN {X 0,Y 263.326,Z 305.3,A -85,B 0,C 180,E1 -18190.768,E2 -18190.768} C_VEL
LIN {X 0,Y 263.303,Z 305.305,A -85,B 0,C 180,E1 -18195.481,E2 -18195.481} C_VEL
LIN {X 0,Y 263.203,Z 305.288,A -85,B 0,C 180,E1 -18200.312,E2 -18200.312} C_VEL
LIN {X 0,Y 263.18,Z 305.32,A -85,B 0,C 180,E1 -18205.294,E2 -18205.294} C_VEL
LIN {X 0,Y 263.149,Z 305.309,A -85,B 0,C 180,E1 -18208.733,E2 -18208.733} C_VEL
LIN {X 0,Y 263.127,Z 305.327,A -85,B 0,C 180,E1 -18212.289,E2 -18212.289} C_VEL
LIN {X 0,Y 263.176,Z 305.325,A -85,B 0,C 180,E1 -18216.764,E2 -18216.764} C_VEL
LIN {X 0,Y 263.12,Z 305.334,A -85,B 0,C 180,E1 -18221.594,E2 -18221.594} C_VEL
LIN {X 0,Y 263.122,Z 305.332,A -85,B 0,C 180,E1 -18223.126,E2 -18223.126} C_VEL
LIN {X 0,Y 264.153,Z 308.26,A -85,B 0,C 180,E1 -18223.502,E2 -18223.502} C_VEL
LIN {X 0,Y 266.47,Z 310.871,A -85,B 0,C 180,E1 -18224.128,E2 -18224.128} C_VEL
LIN {X 0,Y 268.521,Z 314.067,A -85,B 0,C 180,E1 -18224.701,E2 -18224.701} C_VEL
LIN {X 0,Y 270.083,Z 316.185,A -85,B 0,C 180,E1 -18225.116,E2 -18225.116} C_VEL
LIN {X 0,Y 275.987,Z 324.733,A -85,B 0,C 180,E1 -18226.635,E2 -18226.635} C_VEL
LIN {X 0,Y 283.277,Z 336.131,A -85,B 0,C 180,E1 -18228.403,E2 -18228.403} C_VEL
LIN {X 0,Y 290.812,Z 350.672,A -85,B 0,C 180,E1 -18230.179,E2 -18230.179} C_VEL
LIN {X 0,Y 297.058,Z 364.337,A -85,B 0,C 180,E1 -18231.6,E2 -18231.6} C_VEL
LIN {X 0,Y 293.264,Z 452.175,A -85,B 0,C 180,E1 -18233.675,E2 -18233.675} C_VEL
LIN {X 0,Y 292.219,Z 470.083,A -85,B 0,C 180,E1 -18234.164,E2 -18234.164} C_VEL
LIN {X 0,Y 290.686,Z 485.642,A -85,B 0,C 180,E1 -18234.851,E2 -18234.851} C_VEL
LIN {X 0,Y 288.788,Z 499.971,A -85,B 0,C 180,E1 -18235.753,E2 -18235.753} C_VEL
LIN {X 0,Y 286.592,Z 513.606,A -85,B 0,C 180,E1 -18236.886,E2 -18236.886} C_VEL
LIN {X 0,Y 283.859,Z 526.904,A -85,B 0,C 180,E1 -18238.257,E2 -18238.257} C_VEL
LIN {X 0,Y 281.066,Z 538.926,A -85,B 0,C 180,E1 -18239.788,E2 -18239.788} C_VEL
LIN {X 0,Y 277.844,Z 551.131,A -85,B 0,C 180,E1 -18241.689,E2 -18241.689} C_VEL
LIN {X 0,Y 274.745,Z 562.512,A -85,B 0,C 180,E1 -18243.882,E2 -18243.882} C_VEL
LIN {X 0,Y 271.574,Z 573.032,A -85,B 0,C 180,E1 -18246.352,E2 -18246.352} C_VEL
LIN {X 0,Y 268.847,Z 581.985,A -85,B 0,C 180,E1 -18248.935,E2 -18248.935} C_VEL
LIN {X 0,Y 266.282,Z 590.14,A -85,B 0,C 180,E1 -18251.834,E2 -18251.834} C_VEL
LIN {X 0,Y 264.517,Z 596.327,A -85,B 0,C 180,E1 -18254.592,E2 -18254.592} C_VEL
LIN {X 0,Y 262.999,Z 601.766,A -85,B 0,C 180,E1 -18257.656,E2 -18257.656} C_VEL
LIN {X 0,Y 262.055,Z 605.865,A -85,B 0,C 180,E1 -18260.74,E2 -18260.74} C_VEL
LIN {X 0,Y 261.44,Z 608.744,A -85,B 0,C 180,E1 -18263.827,E2 -18263.827} C_VEL
LIN {X 0,Y 261.222,Z 610.471,A -85,B 0,C 180,E1 -18266.916,E2 -18266.916} C_VEL
LIN {X 0,Y 261.133,Z 611.074,A -85,B 0,C 180,E1 -18270,E2 -18270} C_VEL
LIN {X 0,Y 261.219,Z 610.511,A -85,B 0,C 180,E1 -18273.084,E2 -18273.084} C_VEL
LIN {X 0,Y 261.438,Z 608.836,A -85,B 0,C 180,E1 -18276.173,E2 -18276.173} C_VEL
LIN {X 0,Y 262.003,Z 606.007,A -85,B 0,C 180,E1 -18279.261,E2 -18279.261} C_VEL
LIN {X 0,Y 262.952,Z 601.954,A -85,B 0,C 180,E1 -18282.346,E2 -18282.346} C_VEL
LIN {X 0,Y 264.489,Z 596.574,A -85,B 0,C 180,E1 -18285.409,E2 -18285.409} C_VEL
LIN {X 0,Y 266.472,Z 589.717,A -85,B 0,C 180,E1 -18288.45,E2 -18288.45} C_VEL
LIN {X 0,Y 268.749,Z 582.34,A -85,B 0,C 180,E1 -18291.073,E2 -18291.073} C_VEL
LIN {X 0,Y 271.474,Z 573.445,A -85,B 0,C 180,E1 -18293.657,E2 -18293.657} C_VEL
LIN {X 0,Y 274.236,Z 564.368,A -85,B 0,C 180,E1 -18295.827,E2 -18295.827} C_VEL
LIN {X 0,Y 276.669,Z 555.604,A -85,B 0,C 180,E1 -18297.618,E2 -18297.618} C_VEL
LIN {X 0,Y 279.798,Z 544.3,A -85,B 0,C 180,E1 -18299.533,E2 -18299.533} C_VEL
LIN {X 0,Y 282.809,Z 532.012,A -85,B 0,C 180,E1 -18301.248,E2 -18301.248} C_VEL
LIN {X 0,Y 285.708,Z 518.572,A -85,B 0,C 180,E1 -18302.762,E2 -18302.762} C_VEL
LIN {X 0,Y 288.071,Z 505.33,A -85,B 0,C 180,E1 -18303.953,E2 -18303.953} C_VEL
LIN {X 0,Y 290.027,Z 491.625,A -85,B 0,C 180,E1 -18304.923,E2 -18304.923} C_VEL
LIN {X 0,Y 291.703,Z 476.719,A -85,B 0,C 180,E1 -18305.696,E2 -18305.696} C_VEL
LIN {X 0,Y 292.936,Z 461.345,A -85,B 0,C 180,E1 -18306.212,E2 -18306.212} C_VEL
LIN {X 0,Y 297.18,Z 364.389,A -85,B 0,C 180,E1 -18308.509,E2 -18308.509} C_VEL
LIN {X 0,Y 288.97,Z 346.793,A -85,B 0,C 180,E1 -18310.386,E2 -18310.386} C_VEL
LIN {X 0,Y 282.008,Z 333.932,A -85,B 0,C 180,E1 -18312.04,E2 -18312.04} C_VEL
LIN {X 0,Y 273.919,Z 321.706,A -85,B 0,C 180,E1 -18314.031,E2 -18314.031} C_VEL
LIN {X 0,Y 271.494,Z 318.234,A -85,B 0,C 180,E1 -18314.657,E2 -18314.657} C_VEL
LIN {X 0,Y 268.979,Z 314.545,A -85,B 0,C 180,E1 -18315.33,E2 -18315.33} C_VEL
LIN {X 0,Y 266.679,Z 311.33,A -85,B 0,C 180,E1 -18315.958,E2 -18315.958} C_VEL
LIN {X 0,Y 265.857,Z 310.099,A -85,B 0,C 180,E1 -18316.189,E2 -18316.189} C_VEL
LIN {X 0,Y 263.947,Z 307.828,A -85,B 0,C 180,E1 -18316.714,E2 -18316.714} C_VEL
LIN {X 0,Y 263.116,Z 305.322,A -85,B 0,C 180,E1 -18317.036,E2 -18317.036} C_VEL
LIN {X 0,Y 263.107,Z 305.326,A -85,B 0,C 180,E1 -18321.425,E2 -18321.425} C_VEL
LIN {X 0,Y 263.153,Z 305.307,A -85,B 0,C 180,E1 -18324.016,E2 -18324.016} C_VEL
LIN {X 0,Y 263.114,Z 305.311,A -85,B 0,C 180,E1 -18328.049,E2 -18328.049} C_VEL
LIN {X 0,Y 262.434,Z 305.391,A -85,B 0,C 180,E1 -18329.327,E2 -18329.327} C_VEL
LIN {X 0,Y 259.564,Z 305.765,A -85,B 0,C 180,E1 -18331.41,E2 -18331.41} C_VEL
LIN {X 0,Y 257.174,Z 306.075,A -85,B 0,C 180,E1 -18333.105,E2 -18333.105} C_VEL
LIN {X 0,Y 256.207,Z 306.188,A -85,B 0,C 180,E1 -18334.419,E2 -18334.419} C_VEL
LIN {X 0,Y 256.16,Z 306.194,A -85,B 0,C 180,E1 -18334.864,E2 -18334.864} C_VEL
LIN {X 0,Y 256.141,Z 306.197,A -85,B 0,C 180,E1 -18339.103,E2 -18339.103} C_VEL
LIN {X 0,Y 256.238,Z 306.191,A -85,B 0,C 180,E1 -18344.081,E2 -18344.081} C_VEL
LIN {X 0,Y 256.283,Z 306.187,A -85,B 0,C 180,E1 -18348.933,E2 -18348.933} C_VEL
LIN {X 0,Y 256.49,Z 306.155,A -85,B 0,C 180,E1 -18352.125,E2 -18352.125} C_VEL
LIN {X 0,Y 256.454,Z 306.159,A -85,B 0,C 180,E1 -18356.858,E2 -18356.858} C_VEL
LIN {X 0,Y 256.734,Z 306.118,A -85,B 0,C 180,E1 -18360,E2 -18360} C_VEL
LIN {X 0,Y 256.445,Z 306.164,A -85,B 0,C 180,E1 -18363.142,E2 -18363.142} C_VEL
LIN {X 0,Y 256.487,Z 306.158,A -85,B 0,C 180,E1 -18367.874,E2 -18367.874} C_VEL
LIN {X 0,Y 256.282,Z 306.189,A -85,B 0,C 180,E1 -18371.067,E2 -18371.067} C_VEL
LIN {X 0,Y 256.223,Z 306.198,A -85,B 0,C 180,E1 -18375.92,E2 -18375.92} C_VEL
LIN {X 0,Y 256.114,Z 306.205,A -85,B 0,C 180,E1 -18380.899,E2 -18380.899} C_VEL
LIN {X 0,Y 256.08,Z 306.207,A -85,B 0,C 180,E1 -18385.09,E2 -18385.09} C_VEL
LIN {X 0,Y 256.081,Z 306.211,A -85,B 0,C 180,E1 -18388.574,E2 -18388.574} C_VEL
LIN {X 0,Y 256.068,Z 306.214,A -85,B 0,C 180,E1 -18391.702,E2 -18391.702} C_VEL
LIN {X 0,Y 256.073,Z 306.211,A -85,B 0,C 180,E1 -18395.194,E2 -18395.194} C_VEL
LIN {X 0,Y 256.043,Z 306.232,A -85,B 0,C 180,E1 -18398.894,E2 -18398.894} C_VEL
LIN {X 0,Y 258.123,Z 312.448,A -85,B 0,C 180,E1 -18401.718,E2 -18401.718} C_VEL
LIN {X 0,Y 261.306,Z 317.391,A -85,B 0,C 180,E1 -18402.686,E2 -18402.686} C_VEL
LIN {X 0,Y 266.222,Z 325.326,A -85,B 0,C 180,E1 -18404.115,E2 -18404.115} C_VEL
LIN {X 0,Y 272.335,Z 335.62,A -85,B 0,C 180,E1 -18405.789,E2 -18405.789} C_VEL
LIN {X 0,Y 278.731,Z 347.482,A -85,B 0,C 180,E1 -18407.453,E2 -18407.453} C_VEL
LIN {X 0,Y 285.225,Z 360.894,A -85,B 0,C 180,E1 -18409.07,E2 -18409.07} C_VEL
LIN {X 0,Y 291.216,Z 375.019,A -85,B 0,C 180,E1 -18410.521,E2 -18410.521} C_VEL
LIN {X 0,Y 287.567,Z 457.515,A -85,B 0,C 180,E1 -18412.506,E2 -18412.506} C_VEL
LIN {X 0,Y 286.223,Z 481.753,A -85,B 0,C 180,E1 -18413.128,E2 -18413.128} C_VEL
LIN {X 0,Y 284.629,Z 497.124,A -85,B 0,C 180,E1 -18413.769,E2 -18413.769} C_VEL
LIN {X 0,Y 282.423,Z 511.998,A -85,B 0,C 180,E1 -18414.651,E2 -18414.651} C_VEL
LIN {X 0,Y 279.782,Z 526.412,A -85,B 0,C 180,E1 -18415.803,E2 -18415.803} C_VEL
LIN {X 0,Y 277.382,Z 537.777,A -85,B 0,C 180,E1 -18416.952,E2 -18416.952} C_VEL
LIN {X 0,Y 274.231,Z 550.51,A -85,B 0,C 180,E1 -18418.523,E2 -18418.523} C_VEL
LIN {X 0,Y 270.75,Z 563.156,A -85,B 0,C 180,E1 -18420.45,E2 -18420.45} C_VEL
LIN {X 0,Y 267.358,Z 574.652,A -85,B 0,C 180,E1 -18422.612,E2 -18422.612} C_VEL
LIN {X 0,Y 264.397,Z 584.334,A -85,B 0,C 180,E1 -18424.831,E2 -18424.831} C_VEL
LIN {X 0,Y 261.93,Z 592.613,A -85,B 0,C 180,E1 -18427.105,E2 -18427.105} C_VEL
LIN {X 0,Y 259.327,Z 600.768,A -85,B 0,C 180,E1 -18429.786,E2 -18429.786} C_VEL
LIN {X 0,Y 257.001,Z 608.892,A -85,B 0,C 180,E1 -18433.159,E2 -18433.159} C_VEL
LIN {X 0,Y 255.426,Z 615.087,A -85,B 0,C 180,E1 -18436.475,E2 -18436.475} C_VEL
LIN {X 0,Y 254.642,Z 618.591,A -85,B 0,C 180,E1 -18438.861,E2 -18438.861} C_VEL
LIN {X 0,Y 254.125,Z 622.138,A -85,B 0,C 180,E1 -18442.052,E2 -18442.052} C_VEL
LIN {X 0,Y 253.932,Z 624.473,A -85,B 0,C 180,E1 -18445.237,E2 -18445.237} C_VEL
LIN {X 0,Y 254.014,Z 625.65,A -85,B 0,C 180,E1 -18448.415,E2 -18448.415} C_VEL
LIN {X 0,Y 254.053,Z 625.805,A -85,B 0,C 180,E1 -18450,E2 -18450} C_VEL
LIN {X 0,Y 253.937,Z 625.192,A -85,B 0,C 180,E1 -18453.173,E2 -18453.173} C_VEL
LIN {X 0,Y 253.957,Z 623.424,A -85,B 0,C 180,E1 -18456.355,E2 -18456.355} C_VEL
LIN {X 0,Y 254.318,Z 620.481,A -85,B 0,C 180,E1 -18459.544,E2 -18459.544} C_VEL
LIN {X 0,Y 255.12,Z 616.296,A -85,B 0,C 180,E1 -18462.731,E2 -18462.731} C_VEL
LIN {X 0,Y 256.407,Z 610.759,A -85,B 0,C 180,E1 -18465.908,E2 -18465.908} C_VEL
LIN {X 0,Y 258.413,Z 603.726,A -85,B 0,C 180,E1 -18469.048,E2 -18469.048} C_VEL
LIN {X 0,Y 261.08,Z 594.983,A -85,B 0,C 180,E1 -18472.139,E2 -18472.139} C_VEL
LIN {X 0,Y 263.617,Z 587.156,A -85,B 0,C 180,E1 -18474.407,E2 -18474.407} C_VEL
LIN {X 0,Y 266.838,Z 576.273,A -85,B 0,C 180,E1 -18477.021,E2 -18477.021} C_VEL
LIN {X 0,Y 270.463,Z 564.049,A -85,B 0,C 180,E1 -18479.37,E2 -18479.37} C_VEL
LIN {X 0,Y 273.872,Z 551.586,A -85,B 0,C 180,E1 -18481.308,E2 -18481.308} C_VEL
LIN {X 0,Y 276.936,Z 539.353,A -85,B 0,C 180,E1 -18482.846,E2 -18482.846} C_VEL
LIN {X 0,Y 279.755,Z 526.088,A -85,B 0,C 180,E1 -18484.2,E2 -18484.2} C_VEL
LIN {X 0,Y 282.362,Z 511.598,A -85,B 0,C 180,E1 -18485.358,E2 -18485.358} C_VEL
LIN {X 0,Y 284.589,Z 496.589,A -85,B 0,C 180,E1 -18486.237,E2 -18486.237} C_VEL
LIN {X 0,Y 286.082,Z 482.072,A -85,B 0,C 180,E1 -18486.838,E2 -18486.838} C_VEL
LIN {X 0,Y 287.387,Z 459.791,A -85,B 0,C 180,E1 -18487.411,E2 -18487.411} C_VEL
LIN {X 0,Y 291.176,Z 375.384,A -85,B 0,C 180,E1 -18489.433,E2 -18489.433} C_VEL
LIN {X 0,Y 289.896,Z 371.767,A -85,B 0,C 180,E1 -18489.753,E2 -18489.753} C_VEL
LIN {X 0,Y 282.972,Z 356.06,A -85,B 0,C 180,E1 -18491.437,E2 -18491.437} C_VEL
LIN {X 0,Y 275.289,Z 340.907,A -85,B 0,C 180,E1 -18493.382,E2 -18493.382} C_VEL
LIN {X 0,Y 267.505,Z 327.299,A -85,B 0,C 180,E1 -18495.472,E2 -18495.472} C_VEL
LIN {X 0,Y 260.773,Z 316.717,A -85,B 0,C 180,E1 -18497.403,E2 -18497.403} C_VEL
LIN {X 0,Y 257.992,Z 312.117,A -85,B 0,C 180,E1 -18498.273,E2 -18498.273} C_VEL
LIN {X 0,Y 256.042,Z 306.215,A -85,B 0,C 180,E1 -18501.106,E2 -18501.106} C_VEL
LIN {X 0,Y 256.072,Z 306.206,A -85,B 0,C 180,E1 -18504.806,E2 -18504.806} C_VEL
LIN {X 0,Y 256.076,Z 306.212,A -85,B 0,C 180,E1 -18508.57,E2 -18508.57} C_VEL
LIN {X 0,Y 256.074,Z 306.208,A -85,B 0,C 180,E1 -18512.188,E2 -18512.188} C_VEL
LIN {X 0,Y 256.078,Z 306.206,A -85,B 0,C 180,E1 -18515.69,E2 -18515.69} C_VEL
LIN {X 0,Y 256.114,Z 306.192,A -85,B 0,C 180,E1 -18519.101,E2 -18519.101} C_VEL
LIN {X 0,Y 256.223,Z 306.192,A -85,B 0,C 180,E1 -18524.08,E2 -18524.08} C_VEL
LIN {X 0,Y 256.27,Z 306.147,A -85,B 0,C 180,E1 -18528.932,E2 -18528.932} C_VEL
LIN {X 0,Y 256.449,Z 306.166,A -85,B 0,C 180,E1 -18532.124,E2 -18532.124} C_VEL
LIN {X 0,Y 256.444,Z 306.167,A -85,B 0,C 180,E1 -18536.858,E2 -18536.858} C_VEL
LIN {X 0,Y 256.692,Z 306.125,A -85,B 0,C 180,E1 -18538.431,E2 -18538.431} C_VEL
LIN {X 0,Y 256.689,Z 306.131,A -85,B 0,C 180,E1 -18541.569,E2 -18541.569} C_VEL
LIN {X 0,Y 256.443,Z 306.157,A -85,B 0,C 180,E1 -18546.696,E2 -18546.696} C_VEL
LIN {X 0,Y 256.395,Z 306.171,A -85,B 0,C 180,E1 -18549.466,E2 -18549.466} C_VEL
LIN {X 0,Y 256.224,Z 306.187,A -85,B 0,C 180,E1 -18554.292,E2 -18554.292} C_VEL
LIN {X 0,Y 256.156,Z 306.199,A -85,B 0,C 180,E1 -18557.566,E2 -18557.566} C_VEL
LIN {X 0,Y 256.117,Z 306.171,A -85,B 0,C 180,E1 -18561.1,E2 -18561.1} C_VEL
LIN {X 0,Y 256.161,Z 306.195,A -85,B 0,C 180,E1 -18565.128,E2 -18565.128} C_VEL
LIN {X 0,Y 256.094,Z 306.201,A -85,B 0,C 180,E1 -18569.602,E2 -18569.602} C_VEL
LIN {X 0,Y 256.063,Z 306.214,A -85,B 0,C 180,E1 -18573.294,E2 -18573.294} C_VEL
LIN {X 0,Y 256.109,Z 306.202,A -85,B 0,C 180,E1 -18577.271,E2 -18577.271} C_VEL
LIN {X 0,Y 256.08,Z 306.262,A -85,B 0,C 180,E1 -18581.465,E2 -18581.465} C_VEL
LIN {X 0,Y 257.018,Z 308.923,A -85,B 0,C 180,E1 -18581.813,E2 -18581.813} C_VEL
LIN {X 0,Y 259.033,Z 311.128,A -85,B 0,C 180,E1 -18582.402,E2 -18582.402} C_VEL
LIN {X 0,Y 261.928,Z 315.365,A -85,B 0,C 180,E1 -18583.263,E2 -18583.263} C_VEL
LIN {X 0,Y 263.265,Z 317.19,A -85,B 0,C 180,E1 -18583.645,E2 -18583.645} C_VEL
LIN {X 0,Y 269.506,Z 326.148,A -85,B 0,C 180,E1 -18585.36,E2 -18585.36} C_VEL
LIN {X 0,Y 276.626,Z 337.016,A -85,B 0,C 180,E1 -18587.189,E2 -18587.189} C_VEL
LIN {X 0,Y 281.327,Z 345.285,A -85,B 0,C 180,E1 -18588.355,E2 -18588.355} C_VEL
LIN {X 0,Y 288.853,Z 360.628,A -85,B 0,C 180,E1 -18590.169,E2 -18590.169} C_VEL
LIN {X 0,Y 291.433,Z 366.499,A -85,B 0,C 180,E1 -18590.778,E2 -18590.778} C_VEL
LIN {X 0,Y 288.393,Z 434.75,A -85,B 0,C 180,E1 -18592.418,E2 -18592.418} C_VEL
LIN {X 0,Y 286.689,Z 468.021,A -85,B 0,C 180,E1 -18593.253,E2 -18593.253} C_VEL
LIN {X 0,Y 285.258,Z 482.813,A -85,B 0,C 180,E1 -18593.861,E2 -18593.861} C_VEL
LIN {X 0,Y 283.332,Z 497.931,A -85,B 0,C 180,E1 -18594.782,E2 -18594.782} C_VEL
LIN {X 0,Y 281.063,Z 511.728,A -85,B 0,C 180,E1 -18595.893,E2 -18595.893} C_VEL
LIN {X 0,Y 278.213,Z 525.685,A -85,B 0,C 180,E1 -18597.32,E2 -18597.32} C_VEL
LIN {X 0,Y 275.222,Z 537.891,A -85,B 0,C 180,E1 -18598.863,E2 -18598.863} C_VEL
LIN {X 0,Y 272.218,Z 549.234,A -85,B 0,C 180,E1 -18600.625,E2 -18600.625} C_VEL
LIN {X 0,Y 268.937,Z 560.265,A -85,B 0,C 180,E1 -18602.686,E2 -18602.686} C_VEL
LIN {X 0,Y 266.487,Z 568.838,A -85,B 0,C 180,E1 -18604.625,E2 -18604.625} C_VEL
LIN {X 0,Y 263.355,Z 578.533,A -85,B 0,C 180,E1 -18607.236,E2 -18607.236} C_VEL
LIN {X 0,Y 260.699,Z 586.61,A -85,B 0,C 180,E1 -18609.897,E2 -18609.897} C_VEL
LIN {X 0,Y 258.558,Z 593.27,A -85,B 0,C 180,E1 -18612.603,E2 -18612.603} C_VEL
LIN {X 0,Y 256.703,Z 599.43,A -85,B 0,C 180,E1 -18615.736,E2 -18615.736} C_VEL
LIN {X 0,Y 255.456,Z 604.18,A -85,B 0,C 180,E1 -18618.897,E2 -18618.897} C_VEL
LIN {X 0,Y 254.691,Z 607.655,A -85,B 0,C 180,E1 -18622.07,E2 -18622.07} C_VEL
LIN {X 0,Y 254.211,Z 609.952,A -85,B 0,C 180,E1 -18625.243,E2 -18625.243} C_VEL
LIN {X 0,Y 254.085,Z 611.12,A -85,B 0,C 180,E1 -18628.415,E2 -18628.415} C_VEL
LIN {X 0,Y 254.084,Z 611.133,A -85,B 0,C 180,E1 -18631.585,E2 -18631.585} C_VEL
LIN {X 0,Y 254.205,Z 610.017,A -85,B 0,C 180,E1 -18634.758,E2 -18634.758} C_VEL
LIN {X 0,Y 254.61,Z 607.773,A -85,B 0,C 180,E1 -18637.933,E2 -18637.933} C_VEL
LIN {X 0,Y 255.425,Z 604.341,A -85,B 0,C 180,E1 -18641.104,E2 -18641.104} C_VEL
LIN {X 0,Y 256.677,Z 599.642,A -85,B 0,C 180,E1 -18644.266,E2 -18644.266} C_VEL
LIN {X 0,Y 258.546,Z 593.547,A -85,B 0,C 180,E1 -18647.398,E2 -18647.398} C_VEL
LIN {X 0,Y 260.979,Z 585.867,A -85,B 0,C 180,E1 -18650.492,E2 -18650.492} C_VEL
LIN {X 0,Y 263.683,Z 577.674,A -85,B 0,C 180,E1 -18653.149,E2 -18653.149} C_VEL
LIN {X 0,Y 266.904,Z 567.798,A -85,B 0,C 180,E1 -18655.751,E2 -18655.751} C_VEL
LIN {X 0,Y 269.832,Z 557.676,A -85,B 0,C 180,E1 -18657.957,E2 -18657.957} C_VEL
LIN {X 0,Y 273.025,Z 546.674,A -85,B 0,C 180,E1 -18659.916,E2 -18659.916} C_VEL
LIN {X 0,Y 276.084,Z 534.794,A -85,B 0,C 180,E1 -18661.669,E2 -18661.669} C_VEL
LIN {X 0,Y 279.071,Z 521.928,A -85,B 0,C 180,E1 -18663.211,E2 -18663.211} C_VEL
LIN {X 0,Y 281.874,Z 507.342,A -85,B 0,C 180,E1 -18664.607,E2 -18664.607} C_VEL
LIN {X 0,Y 284.055,Z 493.117,A -85,B 0,C 180,E1 -18665.659,E2 -18665.659} C_VEL
LIN {X 0,Y 285.882,Z 477.823,A -85,B 0,C 180,E1 -18666.484,E2 -18666.484} C_VEL
LIN {X 0,Y 287.132,Z 463.031,A -85,B 0,C 180,E1 -18667.01,E2 -18667.01} C_VEL
LIN {X 0,Y 291.557,Z 366.578,A -85,B 0,C 180,E1 -18669.331,E2 -18669.331} C_VEL
LIN {X 0,Y 282.811,Z 347.967,A -85,B 0,C 180,E1 -18671.424,E2 -18671.424} C_VEL
LIN {X 0,Y 277.499,Z 338.315,A -85,B 0,C 180,E1 -18672.738,E2 -18672.738} C_VEL
LIN {X 0,Y 269.832,Z 326.58,A -85,B 0,C 180,E1 -18674.701,E2 -18674.701} C_VEL
LIN {X 0,Y 264.74,Z 319.287,A -85,B 0,C 180,E1 -18676.089,E2 -18676.089} C_VEL
LIN {X 0,Y 261.946,Z 315.371,A -85,B 0,C 180,E1 -18676.886,E2 -18676.886} C_VEL
LIN {X 0,Y 259.798,Z 312.271,A -85,B 0,C 180,E1 -18677.522,E2 -18677.522} C_VEL
LIN {X 0,Y 259.03,Z 311.122,A -85,B 0,C 180,E1 -18677.756,E2 -18677.756} C_VEL
LIN {X 0,Y 257.016,Z 308.909,A -85,B 0,C 180,E1 -18678.347,E2 -18678.347} C_VEL
LIN {X 0,Y 256.075,Z 306.192,A -85,B 0,C 180,E1 -18678.747,E2 -18678.747} C_VEL
LIN {X 0,Y 256.115,Z 306.181,A -85,B 0,C 180,E1 -18682.865,E2 -18682.865} C_VEL
LIN {X 0,Y 256.061,Z 306.211,A -85,B 0,C 180,E1 -18686.706,E2 -18686.706} C_VEL
LIN {X 0,Y 256.059,Z 306.186,A -85,B 0,C 180,E1 -18690.393,E2 -18690.393} C_VEL
LIN {X 0,Y 256.116,Z 306.2,A -85,B 0,C 180,E1 -18693.956,E2 -18693.956} C_VEL
LIN {X 0,Y 256.16,Z 306.194,A -85,B 0,C 180,E1 -18694.864,E2 -18694.864} C_VEL
LIN {X 0,Y 255.896,Z 306.233,A -85,B 0,C 180,E1 -18695.741,E2 -18695.741} C_VEL
LIN {X 0,Y 254.559,Z 306.402,A -85,B 0,C 180,E1 -18697.036,E2 -18697.036} C_VEL
LIN {X 0,Y 250.167,Z 306.948,A -85,B 0,C 180,E1 -18700.05,E2 -18700.05} C_VEL
LIN {X 0,Y 249.151,Z 307.068,A -85,B 0,C 180,E1 -18701.402,E2 -18701.402} C_VEL
LIN {X 0,Y 249.097,Z 307.071,A -85,B 0,C 180,E1 -18701.859,E2 -18701.859} C_VEL
LIN {X 0,Y 249.168,Z 307.069,A -85,B 0,C 180,E1 -18705.294,E2 -18705.294} C_VEL
LIN {X 0,Y 249.379,Z 307.036,A -85,B 0,C 180,E1 -18710.519,E2 -18710.519} C_VEL
LIN {X 0,Y 249.429,Z 307.04,A -85,B 0,C 180,E1 -18713.529,E2 -18713.529} C_VEL
LIN {X 0,Y 249.657,Z 307.011,A -85,B 0,C 180,E1 -18718.387,E2 -18718.387} C_VEL
LIN {X 0,Y 249.653,Z 307.01,A -85,B 0,C 180,E1 -18721.613,E2 -18721.613} C_VEL
LIN {X 0,Y 249.425,Z 307.04,A -85,B 0,C 180,E1 -18726.471,E2 -18726.471} C_VEL
LIN {X 0,Y 249.336,Z 307.042,A -85,B 0,C 180,E1 -18729.737,E2 -18729.737} C_VEL
LIN {X 0,Y 249.163,Z 307.069,A -85,B 0,C 180,E1 -18734.706,E2 -18734.706} C_VEL
LIN {X 0,Y 249.087,Z 307.074,A -85,B 0,C 180,E1 -18738.081,E2 -18738.081} C_VEL
LIN {X 0,Y 249.036,Z 307.082,A -85,B 0,C 180,E1 -18741.523,E2 -18741.523} C_VEL
LIN {X 0,Y 249.042,Z 307.081,A -85,B 0,C 180,E1 -18745.442,E2 -18745.442} C_VEL
LIN {X 0,Y 249.028,Z 307.09,A -85,B 0,C 180,E1 -18748.973,E2 -18748.973} C_VEL
LIN {X 0,Y 249.022,Z 307.083,A -85,B 0,C 180,E1 -18752.427,E2 -18752.427} C_VEL
LIN {X 0,Y 249.069,Z 307.079,A -85,B 0,C 180,E1 -18757.111,E2 -18757.111} C_VEL
LIN {X 0,Y 249.061,Z 307.155,A -85,B 0,C 180,E1 -18757.384,E2 -18757.384} C_VEL
LIN {X 0,Y 250.663,Z 312.044,A -85,B 0,C 180,E1 -18759.762,E2 -18759.762} C_VEL
LIN {X 0,Y 253.898,Z 316.955,A -85,B 0,C 180,E1 -18760.834,E2 -18760.834} C_VEL
LIN {X 0,Y 261.52,Z 328.951,A -85,B 0,C 180,E1 -18763.191,E2 -18763.191} C_VEL
LIN {X 0,Y 268.053,Z 340.13,A -85,B 0,C 180,E1 -18765.064,E2 -18765.064} C_VEL
LIN {X 0,Y 274.565,Z 352.439,A -85,B 0,C 180,E1 -18766.829,E2 -18766.829} C_VEL
LIN {X 0,Y 281.812,Z 367.757,A -85,B 0,C 180,E1 -18768.698,E2 -18768.698} C_VEL
LIN {X 0,Y 285.724,Z 377.266,A -85,B 0,C 180,E1 -18769.686,E2 -18769.686} C_VEL
LIN {X 0,Y 281.078,Z 474.708,A -85,B 0,C 180,E1 -18772.054,E2 -18772.054} C_VEL
LIN {X 0,Y 279.742,Z 490.007,A -85,B 0,C 180,E1 -18772.58,E2 -18772.58} C_VEL
LIN {X 0,Y 277.653,Z 505.56,A -85,B 0,C 180,E1 -18773.387,E2 -18773.387} C_VEL
LIN {X 0,Y 275.052,Z 520.437,A -85,B 0,C 180,E1 -18774.459,E2 -18774.459} C_VEL
LIN {X 0,Y 272.15,Z 534.102,A -85,B 0,C 180,E1 -18775.744,E2 -18775.744} C_VEL
LIN {X 0,Y 268.889,Z 547.722,A -85,B 0,C 180,E1 -18777.38,E2 -18777.38} C_VEL
LIN {X 0,Y 265.551,Z 559.736,A -85,B 0,C 180,E1 -18779.152,E2 -18779.152} C_VEL
LIN {X 0,Y 262.134,Z 570.868,A -85,B 0,C 180,E1 -18781.146,E2 -18781.146} C_VEL
LIN {X 0,Y 258.824,Z 581.438,A -85,B 0,C 180,E1 -18783.47,E2 -18783.47} C_VEL
LIN {X 0,Y 255.77,Z 591.152,A -85,B 0,C 180,E1 -18786.091,E2 -18786.091} C_VEL
LIN {X 0,Y 252.974,Z 599.482,A -85,B 0,C 180,E1 -18788.829,E2 -18788.829} C_VEL
LIN {X 0,Y 250.53,Z 607.316,A -85,B 0,C 180,E1 -18792.027,E2 -18792.027} C_VEL
LIN {X 0,Y 248.771,Z 613.556,A -85,B 0,C 180,E1 -18795.271,E2 -18795.271} C_VEL
LIN {X 0,Y 247.61,Z 618.387,A -85,B 0,C 180,E1 -18798.54,E2 -18798.54} C_VEL
LIN {X 0,Y 247.044,Z 621.934,A -85,B 0,C 180,E1 -18801.823,E2 -18801.823} C_VEL
LIN {X 0,Y 246.841,Z 624.324,A -85,B 0,C 180,E1 -18805.21,E2 -18805.21} C_VEL
LIN {X 0,Y 246.921,Z 625.447,A -85,B 0,C 180,E1 -18808.369,E2 -18808.369} C_VEL
LIN {X 0,Y 246.982,Z 625.603,A -85,B 0,C 180,E1 -18810,E2 -18810} C_VEL
LIN {X 0,Y 246.839,Z 624.988,A -85,B 0,C 180,E1 -18813.264,E2 -18813.264} C_VEL
LIN {X 0,Y 246.872,Z 623.22,A -85,B 0,C 180,E1 -18816.538,E2 -18816.538} C_VEL
LIN {X 0,Y 247.275,Z 620.276,A -85,B 0,C 180,E1 -18819.818,E2 -18819.818} C_VEL
LIN {X 0,Y 248.153,Z 616.091,A -85,B 0,C 180,E1 -18823.095,E2 -18823.095} C_VEL
LIN {X 0,Y 249.5,Z 610.552,A -85,B 0,C 180,E1 -18826.36,E2 -18826.36} C_VEL
LIN {X 0,Y 251.655,Z 603.519,A -85,B 0,C 180,E1 -18829.58,E2 -18829.58} C_VEL
LIN {X 0,Y 254.469,Z 594.777,A -85,B 0,C 180,E1 -18832.746,E2 -18832.746} C_VEL
LIN {X 0,Y 257.07,Z 586.947,A -85,B 0,C 180,E1 -18835.071,E2 -18835.071} C_VEL
